    movel(p[x_c + 0.055265, y_c + -0.106909, z_c, rx, ry, rz], a, v)
    movel(p[x_c + 0.055232, y_c + -0.106894, z_c, rx, ry, rz], a, v)
    movel(p[x_c + 0.055195, y_c + -0.106876, z_c, rx, ry, rz], a, v)
    movel(p[x_c + 0.055155, y_c + -0.106856, z_c, rx, ry, rz], a, v)
    movel(p[x_c + 0.055111, y_c + -0.106832, z_c, rx, ry, rz], a, v)
    movel(p[x_c + 0.055063, y_c + -0.106806, z_c, rx, ry, rz], a, v)
    movel(p[x_c + 0.055012, y_c + -0.106778, z_c, rx, ry, rz], a, v)
    movel(p[x_c + 0.054956, y_c + -0.106746, z_c, rx, ry, rz], a, v)
    movel(p[x_c + 0.054897, y_c + -0.106712, z_c, rx, ry, rz], a, v)
    movel(p[x_c + 0.054834, y_c + -0.106675, z_c, rx, ry, rz], a, v)
    movel(p[x_c + 0.054767, y_c + -0.106635, z_c, rx, ry, rz], a, v)
    movel(p[x_c + 0.054696, y_c + -0.106592, z_c, rx, ry, rz], a, v)
    movel(p[x_c + 0.054696, y_c + -0.106592, z_c, rx, ry, rz], a, v)
    movel(p[x_c + 0.054632, y_c + -0.106555, z_c, rx, ry, rz], a, v)
    movel(p[x_c + 0.054557, y_c + -0.106511, z_c, rx, ry, rz], a, v)
    movel(p[x_c + 0.054470, y_c + -0.106462, z_c, rx, ry, rz], a, v)
    movel(p[x_c + 0.054372, y_c + -0.106408, z_c, rx, ry, rz], a, v)
    movel(p[x_c + 0.054263, y_c + -0.106348, z_c, rx, ry, rz], a, v)
    movel(p[x_c + 0.054144, y_c + -0.106284, z_c, rx, ry, rz], a, v)
    movel(p[x_c + 0.054016, y_c + -0.106215, z_c, rx, ry, rz], a, v)
    movel(p[x_c + 0.053879, y_c + -0.106142, z_c, rx, ry, rz], a, v)
    movel(p[x_c + 0.053733, y_c + -0.106065, z_c, rx, ry, rz], a, v)
    movel(p[x_c + 0.053580, y_c + -0.105984, z_c, rx, ry, rz], a, v)
    movel(p[x_c + 0.053420, y_c + -0.105900, z_c, rx, ry, rz], a, v)
    movel(p[x_c + 0.053253, y_c + -0.105813, z_c, rx, ry, rz], a, v)
    movel(p[x_c + 0.053080, y_c + -0.105722, z_c, rx, ry, rz], a, v)
    movel(p[x_c + 0.052901, y_c + -0.105630, z_c, rx, ry, rz], a, v)
    movel(p[x_c + 0.052717, y_c + -0.105535, z_c, rx, ry, rz], a, v)
    movel(p[x_c + 0.052529, y_c + -0.105438, z_c, rx, ry, rz], a, v)
    movel(p[x_c + 0.052338, y_c + -0.105339, z_c, rx, ry, rz], a, v)
    movel(p[x_c + 0.052143, y_c + -0.105239, z_c, rx, ry, rz], a, v)
    movel(p[x_c + 0.051945, y_c + -0.105138, z_c, rx, ry, rz], a, v)
    movel(p[x_c + 0.051745, y_c + -0.105036, z_c, rx, ry, rz], a, v)
    movel(p[x_c + 0.051543, y_c + -0.104933, z_c, rx, ry, rz], a, v)
    movel(p[x_c + 0.051341, y_c + -0.104830, z_c, rx, ry, rz], a, v)
    movel(p[x_c + 0.051138, y_c + -0.104727, z_c, rx, ry, rz], a, v)
    movel(p[x_c + 0.050935, y_c + -0.104625, z_c, rx, ry, rz], a, v)
    movel(p[x_c + 0.050733, y_c + -0.104523, z_c, rx, ry, rz], a, v)
    movel(p[x_c + 0.050532, y_c + -0.104421, z_c, rx, ry, rz], a, v)
    movel(p[x_c + 0.050332, y_c + -0.104321, z_c, rx, ry, rz], a, v)
    movel(p[x_c + 0.050135, y_c + -0.104222, z_c, rx, ry, rz], a, v)
    movel(p[x_c + 0.049941, y_c + -0.104125, z_c, rx, ry, rz], a, v)
    movel(p[x_c + 0.049751, y_c + -0.104030, z_c, rx, ry, rz], a, v)
    movel(p[x_c + 0.049564, y_c + -0.103938, z_c, rx, ry, rz], a, v)
    movel(p[x_c + 0.049382, y_c + -0.103847, z_c, rx, ry, rz], a, v)
    movel(p[x_c + 0.049205, y_c + -0.103760, z_c, rx, ry, rz], a, v)
    movel(p[x_c + 0.049034, y_c + -0.103676, z_c, rx, ry, rz], a, v)
    movel(p[x_c + 0.048869, y_c + -0.103595, z_c, rx, ry, rz], a, v)
    movel(p[x_c + 0.048711, y_c + -0.103517, z_c, rx, ry, rz], a, v)
    movel(p[x_c + 0.048560, y_c + -0.103444, z_c, rx, ry, rz], a, v)
    movel(p[x_c + 0.048417, y_c + -0.103375, z_c, rx, ry, rz], a, v)
    movel(p[x_c + 0.048283, y_c + -0.103310, z_c, rx, ry, rz], a, v)
    movel(p[x_c + 0.048158, y_c + -0.103251, z_c, rx, ry, rz], a, v)
    movel(p[x_c + 0.048042, y_c + -0.103196, z_c, rx, ry, rz], a, v)
    movel(p[x_c + 0.047937, y_c + -0.103147, z_c, rx, ry, rz], a, v)
    movel(p[x_c + 0.047842, y_c + -0.103103, z_c, rx, ry, rz], a, v)
    movel(p[x_c + 0.047759, y_c + -0.103065, z_c, rx, ry, rz], a, v)
    movel(p[x_c + 0.047687, y_c + -0.103034, z_c, rx, ry, rz], a, v)
    movel(p[x_c + 0.047628, y_c + -0.103009, z_c, rx, ry, rz], a, v)
    movel(p[x_c + 0.047582, y_c + -0.102991, z_c, rx, ry, rz], a, v)
    movel(p[x_c + 0.047550, y_c + -0.102980, z_c, rx, ry, rz], a, v)
    movel(p[x_c + 0.047531, y_c + -0.102976, z_c, rx, ry, rz], a, v)
    movel(p[x_c + 0.047531, y_c + -0.102976, z_c, rx, ry, rz], a, v)
    movel(p[x_c + 0.047525, y_c + -0.102977, z_c, rx, ry, rz], a, v)
    movel(p[x_c + 0.047514, y_c + -0.102981, z_c, rx, ry, rz], a, v)
    movel(p[x_c + 0.047501, y_c + -0.102987, z_c, rx, ry, rz], a, v)
    movel(p[x_c + 0.047483, y_c + -0.102996, z_c, rx, ry, rz], a, v)
    movel(p[x_c + 0.047462, y_c + -0.103007, z_c, rx, ry, rz], a, v)
    movel(p[x_c + 0.047437, y_c + -0.103020, z_c, rx, ry, rz], a, v)
    movel(p[x_c + 0.047409, y_c + -0.103036, z_c, rx, ry, rz], a, v)
    movel(p[x_c + 0.047378, y_c + -0.103054, z_c, rx, ry, rz], a, v)
    movel(p[x_c + 0.047343, y_c + -0.103074, z_c, rx, ry, rz], a, v)
    movel(p[x_c + 0.047306, y_c + -0.103097, z_c, rx, ry, rz], a, v)
    movel(p[x_c + 0.047265, y_c + -0.103121, z_c, rx, ry, rz], a, v)
    movel(p[x_c + 0.047220, y_c + -0.103148, z_c, rx, ry, rz], a, v)
    movel(p[x_c + 0.047173, y_c + -0.103177, z_c, rx, ry, rz], a, v)
    movel(p[x_c + 0.047123, y_c + -0.103207, z_c, rx, ry, rz], a, v)
    movel(p[x_c + 0.047070, y_c + -0.103240, z_c, rx, ry, rz], a, v)
    movel(p[x_c + 0.047014, y_c + -0.103275, z_c, rx, ry, rz], a, v)
    movel(p[x_c + 0.046956, y_c + -0.103311, z_c, rx, ry, rz], a, v)
    movel(p[x_c + 0.046894, y_c + -0.103350, z_c, rx, ry, rz], a, v)
    movel(p[x_c + 0.046830, y_c + -0.103390, z_c, rx, ry, rz], a, v)
    movel(p[x_c + 0.046763, y_c + -0.103432, z_c, rx, ry, rz], a, v)
    movel(p[x_c + 0.046694, y_c + -0.103476, z_c, rx, ry, rz], a, v)
    movel(p[x_c + 0.046623, y_c + -0.103521, z_c, rx, ry, rz], a, v)
    movel(p[x_c + 0.046548, y_c + -0.103568, z_c, rx, ry, rz], a, v)
    movel(p[x_c + 0.046472, y_c + -0.103617, z_c, rx, ry, rz], a, v)
    movel(p[x_c + 0.046393, y_c + -0.103667, z_c, rx, ry, rz], a, v)
    movel(p[x_c + 0.046312, y_c + -0.103719, z_c, rx, ry, rz], a, v)
    movel(p[x_c + 0.046229, y_c + -0.103773, z_c, rx, ry, rz], a, v)
    movel(p[x_c + 0.046144, y_c + -0.103827, z_c, rx, ry, rz], a, v)
    movel(p[x_c + 0.046057, y_c + -0.103884, z_c, rx, ry, rz], a, v)
    movel(p[x_c + 0.045968, y_c + -0.103941, z_c, rx, ry, rz], a, v)
    movel(p[x_c + 0.045877, y_c + -0.104000, z_c, rx, ry, rz], a, v)
    movel(p[x_c + 0.045784, y_c + -0.104061, z_c, rx, ry, rz], a, v)
    movel(p[x_c + 0.045689, y_c + -0.104122, z_c, rx, ry, rz], a, v)
    movel(p[x_c + 0.045593, y_c + -0.104185, z_c, rx, ry, rz], a, v)
    movel(p[x_c + 0.045495, y_c + -0.104249, z_c, rx, ry, rz], a, v)
    movel(p[x_c + 0.045395, y_c + -0.104314, z_c, rx, ry, rz], a, v)
    movel(p[x_c + 0.045294, y_c + -0.104380, z_c, rx, ry, rz], a, v)
    movel(p[x_c + 0.045191, y_c + -0.104447, z_c, rx, ry, rz], a, v)
    movel(p[x_c + 0.045088, y_c + -0.104515, z_c, rx, ry, rz], a, v)
    movel(p[x_c + 0.044982, y_c + -0.104584, z_c, rx, ry, rz], a, v)
    movel(p[x_c + 0.044876, y_c + -0.104654, z_c, rx, ry, rz], a, v)
    movel(p[x_c + 0.044768, y_c + -0.104725, z_c, rx, ry, rz], a, v)
    movel(p[x_c + 0.044659, y_c + -0.104797, z_c, rx, ry, rz], a, v)
    movel(p[x_c + 0.044549, y_c + -0.104870, z_c, rx, ry, rz], a, v)
    movel(p[x_c + 0.044438, y_c + -0.104943, z_c, rx, ry, rz], a, v)
    movel(p[x_c + 0.044326, y_c + -0.105017, z_c, rx, ry, rz], a, v)
    movel(p[x_c + 0.044213, y_c + -0.105092, z_c, rx, ry, rz], a, v)
    movel(p[x_c + 0.044099, y_c + -0.105168, z_c, rx, ry, rz], a, v)
    movel(p[x_c + 0.043985, y_c + -0.105244, z_c, rx, ry, rz], a, v)
    movel(p[x_c + 0.043985, y_c + -0.105244, z_c, rx, ry, rz], a, v)
    movel(p[x_c + 0.043855, y_c + -0.105330, z_c, rx, ry, rz], a, v)
    movel(p[x_c + 0.043724, y_c + -0.105416, z_c, rx, ry, rz], a, v)
    movel(p[x_c + 0.043591, y_c + -0.105503, z_c, rx, ry, rz], a, v)
    movel(p[x_c + 0.043457, y_c + -0.105590, z_c, rx, ry, rz], a, v)
    movel(p[x_c + 0.043321, y_c + -0.105677, z_c, rx, ry, rz], a, v)
    movel(p[x_c + 0.043184, y_c + -0.105765, z_c, rx, ry, rz], a, v)
    movel(p[x_c + 0.043045, y_c + -0.105853, z_c, rx, ry, rz], a, v)
    movel(p[x_c + 0.042905, y_c + -0.105941, z_c, rx, ry, rz], a, v)
    movel(p[x_c + 0.042764, y_c + -0.106030, z_c, rx, ry, rz], a, v)
    movel(p[x_c + 0.042622, y_c + -0.106119, z_c, rx, ry, rz], a, v)
    movel(p[x_c + 0.042478, y_c + -0.106207, z_c, rx, ry, rz], a, v)
    movel(p[x_c + 0.042334, y_c + -0.106296, z_c, rx, ry, rz], a, v)
    movel(p[x_c + 0.042188, y_c + -0.106385, z_c, rx, ry, rz], a, v)
    movel(p[x_c + 0.042042, y_c + -0.106474, z_c, rx, ry, rz], a, v)
    movel(p[x_c + 0.041894, y_c + -0.106563, z_c, rx, ry, rz], a, v)
    movel(p[x_c + 0.041746, y_c + -0.106652, z_c, rx, ry, rz], a, v)
    movel(p[x_c + 0.041597, y_c + -0.106741, z_c, rx, ry, rz], a, v)
    movel(p[x_c + 0.041447, y_c + -0.106830, z_c, rx, ry, rz], a, v)
    movel(p[x_c + 0.041296, y_c + -0.106919, z_c, rx, ry, rz], a, v)
    movel(p[x_c + 0.041145, y_c + -0.107007, z_c, rx, ry, rz], a, v)
    movel(p[x_c + 0.040994, y_c + -0.107096, z_c, rx, ry, rz], a, v)
    movel(p[x_c + 0.040841, y_c + -0.107184, z_c, rx, ry, rz], a, v)
    movel(p[x_c + 0.040688, y_c + -0.107272, z_c, rx, ry, rz], a, v)
    movel(p[x_c + 0.040535, y_c + -0.107360, z_c, rx, ry, rz], a, v)
    movel(p[x_c + 0.040382, y_c + -0.107447, z_c, rx, ry, rz], a, v)
    movel(p[x_c + 0.040228, y_c + -0.107535, z_c, rx, ry, rz], a, v)
    movel(p[x_c + 0.040074, y_c + -0.107621, z_c, rx, ry, rz], a, v)
    movel(p[x_c + 0.039919, y_c + -0.107708, z_c, rx, ry, rz], a, v)
    movel(p[x_c + 0.039765, y_c + -0.107794, z_c, rx, ry, rz], a, v)
    movel(p[x_c + 0.039610, y_c + -0.107879, z_c, rx, ry, rz], a, v)
    movel(p[x_c + 0.039456, y_c + -0.107964, z_c, rx, ry, rz], a, v)
    movel(p[x_c + 0.039301, y_c + -0.108049, z_c, rx, ry, rz], a, v)
    movel(p[x_c + 0.039147, y_c + -0.108133, z_c, rx, ry, rz], a, v)
    movel(p[x_c + 0.038992, y_c + -0.108216, z_c, rx, ry, rz], a, v)
    movel(p[x_c + 0.038838, y_c + -0.108299, z_c, rx, ry, rz], a, v)
    movel(p[x_c + 0.038684, y_c + -0.108381, z_c, rx, ry, rz], a, v)
    movel(p[x_c + 0.038531, y_c + -0.108463, z_c, rx, ry, rz], a, v)
    movel(p[x_c + 0.038377, y_c + -0.108543, z_c, rx, ry, rz], a, v)
    movel(p[x_c + 0.038224, y_c + -0.108623, z_c, rx, ry, rz], a, v)
    movel(p[x_c + 0.038072, y_c + -0.108703, z_c, rx, ry, rz], a, v)
    movel(p[x_c + 0.037920, y_c + -0.108781, z_c, rx, ry, rz], a, v)
    movel(p[x_c + 0.037769, y_c + -0.108859, z_c, rx, ry, rz], a, v)
    movel(p[x_c + 0.037618, y_c + -0.108936, z_c, rx, ry, rz], a, v)
    movel(p[x_c + 0.037468, y_c + -0.109012, z_c, rx, ry, rz], a, v)
    movel(p[x_c + 0.037318, y_c + -0.109087, z_c, rx, ry, rz], a, v)
    movel(p[x_c + 0.037170, y_c + -0.109161, z_c, rx, ry, rz], a, v)
    movel(p[x_c + 0.037022, y_c + -0.109234, z_c, rx, ry, rz], a, v)
    movel(p[x_c + 0.036875, y_c + -0.109306, z_c, rx, ry, rz], a, v)
    movel(p[x_c + 0.036729, y_c + -0.109377, z_c, rx, ry, rz], a, v)
    movel(p[x_c + 0.036729, y_c + -0.109377, z_c, rx, ry, rz], a, v)
    movel(p[x_c + 0.036600, y_c + -0.109440, z_c, rx, ry, rz], a, v)
    movel(p[x_c + 0.036471, y_c + -0.109503, z_c, rx, ry, rz], a, v)
    movel(p[x_c + 0.036342, y_c + -0.109567, z_c, rx, ry, rz], a, v)
    movel(p[x_c + 0.036213, y_c + -0.109630, z_c, rx, ry, rz], a, v)
    movel(p[x_c + 0.036085, y_c + -0.109694, z_c, rx, ry, rz], a, v)
    movel(p[x_c + 0.035957, y_c + -0.109757, z_c, rx, ry, rz], a, v)
    movel(p[x_c + 0.035830, y_c + -0.109821, z_c, rx, ry, rz], a, v)
    movel(p[x_c + 0.035704, y_c + -0.109885, z_c, rx, ry, rz], a, v)
    movel(p[x_c + 0.035578, y_c + -0.109948, z_c, rx, ry, rz], a, v)
    movel(p[x_c + 0.035453, y_c + -0.110012, z_c, rx, ry, rz], a, v)
    movel(p[x_c + 0.035329, y_c + -0.110075, z_c, rx, ry, rz], a, v)
    movel(p[x_c + 0.035206, y_c + -0.110138, z_c, rx, ry, rz], a, v)
    movel(p[x_c + 0.035085, y_c + -0.110201, z_c, rx, ry, rz], a, v)
    movel(p[x_c + 0.034964, y_c + -0.110263, z_c, rx, ry, rz], a, v)
    movel(p[x_c + 0.034845, y_c + -0.110325, z_c, rx, ry, rz], a, v)
    movel(p[x_c + 0.034727, y_c + -0.110387, z_c, rx, ry, rz], a, v)
    movel(p[x_c + 0.034610, y_c + -0.110448, z_c, rx, ry, rz], a, v)
    movel(p[x_c + 0.034495, y_c + -0.110509, z_c, rx, ry, rz], a, v)
    movel(p[x_c + 0.034382, y_c + -0.110570, z_c, rx, ry, rz], a, v)
    movel(p[x_c + 0.034270, y_c + -0.110629, z_c, rx, ry, rz], a, v)
    movel(p[x_c + 0.034160, y_c + -0.110688, z_c, rx, ry, rz], a, v)
    movel(p[x_c + 0.034052, y_c + -0.110747, z_c, rx, ry, rz], a, v)
    movel(p[x_c + 0.033946, y_c + -0.110804, z_c, rx, ry, rz], a, v)
    movel(p[x_c + 0.033841, y_c + -0.110861, z_c, rx, ry, rz], a, v)
    movel(p[x_c + 0.033739, y_c + -0.110918, z_c, rx, ry, rz], a, v)
    movel(p[x_c + 0.033639, y_c + -0.110973, z_c, rx, ry, rz], a, v)
    movel(p[x_c + 0.033541, y_c + -0.111027, z_c, rx, ry, rz], a, v)
    movel(p[x_c + 0.033446, y_c + -0.111081, z_c, rx, ry, rz], a, v)
    movel(p[x_c + 0.033353, y_c + -0.111133, z_c, rx, ry, rz], a, v)
    movel(p[x_c + 0.033262, y_c + -0.111185, z_c, rx, ry, rz], a, v)
    movel(p[x_c + 0.033174, y_c + -0.111235, z_c, rx, ry, rz], a, v)
    movel(p[x_c + 0.033089, y_c + -0.111284, z_c, rx, ry, rz], a, v)
    movel(p[x_c + 0.033007, y_c + -0.111332, z_c, rx, ry, rz], a, v)
    movel(p[x_c + 0.032927, y_c + -0.111379, z_c, rx, ry, rz], a, v)
    movel(p[x_c + 0.032850, y_c + -0.111425, z_c, rx, ry, rz], a, v)
    movel(p[x_c + 0.032776, y_c + -0.111469, z_c, rx, ry, rz], a, v)
    movel(p[x_c + 0.032705, y_c + -0.111512, z_c, rx, ry, rz], a, v)
    movel(p[x_c + 0.032638, y_c + -0.111554, z_c, rx, ry, rz], a, v)
    movel(p[x_c + 0.032573, y_c + -0.111594, z_c, rx, ry, rz], a, v)
    movel(p[x_c + 0.032512, y_c + -0.111633, z_c, rx, ry, rz], a, v)
    movel(p[x_c + 0.032455, y_c + -0.111670, z_c, rx, ry, rz], a, v)
    movel(p[x_c + 0.032400, y_c + -0.111706, z_c, rx, ry, rz], a, v)
    movel(p[x_c + 0.032350, y_c + -0.111739, z_c, rx, ry, rz], a, v)
    movel(p[x_c + 0.032303, y_c + -0.111772, z_c, rx, ry, rz], a, v)
    movel(p[x_c + 0.032259, y_c + -0.111802, z_c, rx, ry, rz], a, v)
    movel(p[x_c + 0.032220, y_c + -0.111831, z_c, rx, ry, rz], a, v)
    movel(p[x_c + 0.032184, y_c + -0.111858, z_c, rx, ry, rz], a, v)
    movel(p[x_c + 0.032153, y_c + -0.111884, z_c, rx, ry, rz], a, v)
    movel(p[x_c + 0.032125, y_c + -0.111907, z_c, rx, ry, rz], a, v)
    movel(p[x_c + 0.032125, y_c + -0.111907, z_c, rx, ry, rz], a, v)
    movel(p[x_c + 0.032099, y_c + -0.111931, z_c, rx, ry, rz], a, v)
    movel(p[x_c + 0.032070, y_c + -0.111957, z_c, rx, ry, rz], a, v)
    movel(p[x_c + 0.032040, y_c + -0.111986, z_c, rx, ry, rz], a, v)
    movel(p[x_c + 0.032008, y_c + -0.112018, z_c, rx, ry, rz], a, v)
    movel(p[x_c + 0.031974, y_c + -0.112053, z_c, rx, ry, rz], a, v)
    movel(p[x_c + 0.031939, y_c + -0.112089, z_c, rx, ry, rz], a, v)
    movel(p[x_c + 0.031902, y_c + -0.112129, z_c, rx, ry, rz], a, v)
    movel(p[x_c + 0.031863, y_c + -0.112170, z_c, rx, ry, rz], a, v)
    movel(p[x_c + 0.031823, y_c + -0.112214, z_c, rx, ry, rz], a, v)
    movel(p[x_c + 0.031781, y_c + -0.112261, z_c, rx, ry, rz], a, v)
    movel(p[x_c + 0.031737, y_c + -0.112309, z_c, rx, ry, rz], a, v)
    movel(p[x_c + 0.031693, y_c + -0.112360, z_c, rx, ry, rz], a, v)
    movel(p[x_c + 0.031646, y_c + -0.112413, z_c, rx, ry, rz], a, v)
    movel(p[x_c + 0.031599, y_c + -0.112468, z_c, rx, ry, rz], a, v)
    movel(p[x_c + 0.031550, y_c + -0.112524, z_c, rx, ry, rz], a, v)
    movel(p[x_c + 0.031500, y_c + -0.112583, z_c, rx, ry, rz], a, v)
    movel(p[x_c + 0.031449, y_c + -0.112644, z_c, rx, ry, rz], a, v)
    movel(p[x_c + 0.031396, y_c + -0.112706, z_c, rx, ry, rz], a, v)
    movel(p[x_c + 0.031343, y_c + -0.112770, z_c, rx, ry, rz], a, v)
    movel(p[x_c + 0.031289, y_c + -0.112836, z_c, rx, ry, rz], a, v)
    movel(p[x_c + 0.031233, y_c + -0.112903, z_c, rx, ry, rz], a, v)
    movel(p[x_c + 0.031177, y_c + -0.112972, z_c, rx, ry, rz], a, v)
    movel(p[x_c + 0.031119, y_c + -0.113043, z_c, rx, ry, rz], a, v)
    movel(p[x_c + 0.031061, y_c + -0.113114, z_c, rx, ry, rz], a, v)
    movel(p[x_c + 0.031002, y_c + -0.113188, z_c, rx, ry, rz], a, v)
    movel(p[x_c + 0.030942, y_c + -0.113262, z_c, rx, ry, rz], a, v)
    movel(p[x_c + 0.030882, y_c + -0.113338, z_c, rx, ry, rz], a, v)
    movel(p[x_c + 0.030820, y_c + -0.113415, z_c, rx, ry, rz], a, v)
    movel(p[x_c + 0.030759, y_c + -0.113494, z_c, rx, ry, rz], a, v)
    movel(p[x_c + 0.030696, y_c + -0.113573, z_c, rx, ry, rz], a, v)
    movel(p[x_c + 0.030633, y_c + -0.113653, z_c, rx, ry, rz], a, v)
    movel(p[x_c + 0.030570, y_c + -0.113735, z_c, rx, ry, rz], a, v)
    movel(p[x_c + 0.030506, y_c + -0.113817, z_c, rx, ry, rz], a, v)
    movel(p[x_c + 0.030442, y_c + -0.113900, z_c, rx, ry, rz], a, v)
    movel(p[x_c + 0.030377, y_c + -0.113984, z_c, rx, ry, rz], a, v)
    movel(p[x_c + 0.030312, y_c + -0.114069, z_c, rx, ry, rz], a, v)
    movel(p[x_c + 0.030247, y_c + -0.114154, z_c, rx, ry, rz], a, v)
    movel(p[x_c + 0.030182, y_c + -0.114240, z_c, rx, ry, rz], a, v)
    movel(p[x_c + 0.030117, y_c + -0.114326, z_c, rx, ry, rz], a, v)
    movel(p[x_c + 0.030051, y_c + -0.114413, z_c, rx, ry, rz], a, v)
    movel(p[x_c + 0.029986, y_c + -0.114501, z_c, rx, ry, rz], a, v)
    movel(p[x_c + 0.029920, y_c + -0.114588, z_c, rx, ry, rz], a, v)
    movel(p[x_c + 0.029855, y_c + -0.114677, z_c, rx, ry, rz], a, v)
    movel(p[x_c + 0.029789, y_c + -0.114765, z_c, rx, ry, rz], a, v)
    movel(p[x_c + 0.029724, y_c + -0.114854, z_c, rx, ry, rz], a, v)
    movel(p[x_c + 0.029659, y_c + -0.114942, z_c, rx, ry, rz], a, v)
    movel(p[x_c + 0.029594, y_c + -0.115031, z_c, rx, ry, rz], a, v)
    movel(p[x_c + 0.029529, y_c + -0.115120, z_c, rx, ry, rz], a, v)
    movel(p[x_c + 0.029465, y_c + -0.115209, z_c, rx, ry, rz], a, v)
    movel(p[x_c + 0.029465, y_c + -0.115209, z_c, rx, ry, rz], a, v)
    movel(p[x_c + 0.029321, y_c + -0.115407, z_c, rx, ry, rz], a, v)
    movel(p[x_c + 0.029177, y_c + -0.115603, z_c, rx, ry, rz], a, v)
    movel(p[x_c + 0.029032, y_c + -0.115797, z_c, rx, ry, rz], a, v)
    movel(p[x_c + 0.028888, y_c + -0.115988, z_c, rx, ry, rz], a, v)
    movel(p[x_c + 0.028743, y_c + -0.116177, z_c, rx, ry, rz], a, v)
    movel(p[x_c + 0.028599, y_c + -0.116363, z_c, rx, ry, rz], a, v)
    movel(p[x_c + 0.028454, y_c + -0.116547, z_c, rx, ry, rz], a, v)
    movel(p[x_c + 0.028309, y_c + -0.116728, z_c, rx, ry, rz], a, v)
    movel(p[x_c + 0.028165, y_c + -0.116907, z_c, rx, ry, rz], a, v)
    movel(p[x_c + 0.028020, y_c + -0.117083, z_c, rx, ry, rz], a, v)
    movel(p[x_c + 0.027875, y_c + -0.117257, z_c, rx, ry, rz], a, v)
    movel(p[x_c + 0.027730, y_c + -0.117428, z_c, rx, ry, rz], a, v)
    movel(p[x_c + 0.027586, y_c + -0.117597, z_c, rx, ry, rz], a, v)
    movel(p[x_c + 0.027441, y_c + -0.117763, z_c, rx, ry, rz], a, v)
    movel(p[x_c + 0.027296, y_c + -0.117926, z_c, rx, ry, rz], a, v)
    movel(p[x_c + 0.027152, y_c + -0.118087, z_c, rx, ry, rz], a, v)
    movel(p[x_c + 0.027007, y_c + -0.118245, z_c, rx, ry, rz], a, v)
    movel(p[x_c + 0.026863, y_c + -0.118401, z_c, rx, ry, rz], a, v)
    movel(p[x_c + 0.026719, y_c + -0.118554, z_c, rx, ry, rz], a, v)
    movel(p[x_c + 0.026574, y_c + -0.118704, z_c, rx, ry, rz], a, v)
    movel(p[x_c + 0.026430, y_c + -0.118852, z_c, rx, ry, rz], a, v)
    movel(p[x_c + 0.026287, y_c + -0.118997, z_c, rx, ry, rz], a, v)
    movel(p[x_c + 0.026143, y_c + -0.119139, z_c, rx, ry, rz], a, v)
    movel(p[x_c + 0.025999, y_c + -0.119279, z_c, rx, ry, rz], a, v)
    movel(p[x_c + 0.025856, y_c + -0.119415, z_c, rx, ry, rz], a, v)
    movel(p[x_c + 0.025713, y_c + -0.119550, z_c, rx, ry, rz], a, v)
    movel(p[x_c + 0.025570, y_c + -0.119681, z_c, rx, ry, rz], a, v)
    movel(p[x_c + 0.025427, y_c + -0.119810, z_c, rx, ry, rz], a, v)
    movel(p[x_c + 0.025284, y_c + -0.119936, z_c, rx, ry, rz], a, v)
    movel(p[x_c + 0.025142, y_c + -0.120059, z_c, rx, ry, rz], a, v)
    movel(p[x_c + 0.025000, y_c + -0.120179, z_c, rx, ry, rz], a, v)
    movel(p[x_c + 0.024859, y_c + -0.120297, z_c, rx, ry, rz], a, v)
    movel(p[x_c + 0.024717, y_c + -0.120412, z_c, rx, ry, rz], a, v)
    movel(p[x_c + 0.024576, y_c + -0.120524, z_c, rx, ry, rz], a, v)
    movel(p[x_c + 0.024435, y_c + -0.120633, z_c, rx, ry, rz], a, v)
    movel(p[x_c + 0.024295, y_c + -0.120739, z_c, rx, ry, rz], a, v)
    movel(p[x_c + 0.024155, y_c + -0.120842, z_c, rx, ry, rz], a, v)
    movel(p[x_c + 0.024015, y_c + -0.120943, z_c, rx, ry, rz], a, v)
    movel(p[x_c + 0.023875, y_c + -0.121041, z_c, rx, ry, rz], a, v)
    movel(p[x_c + 0.023736, y_c + -0.121135, z_c, rx, ry, rz], a, v)
    movel(p[x_c + 0.023598, y_c + -0.121227, z_c, rx, ry, rz], a, v)
    movel(p[x_c + 0.023459, y_c + -0.121316, z_c, rx, ry, rz], a, v)
    movel(p[x_c + 0.023322, y_c + -0.121402, z_c, rx, ry, rz], a, v)
    movel(p[x_c + 0.023184, y_c + -0.121485, z_c, rx, ry, rz], a, v)
    movel(p[x_c + 0.023047, y_c + -0.121565, z_c, rx, ry, rz], a, v)
    movel(p[x_c + 0.022911, y_c + -0.121642, z_c, rx, ry, rz], a, v)
    movel(p[x_c + 0.022775, y_c + -0.121716, z_c, rx, ry, rz], a, v)
    movel(p[x_c + 0.022639, y_c + -0.121788, z_c, rx, ry, rz], a, v)
    movel(p[x_c + 0.022504, y_c + -0.121856, z_c, rx, ry, rz], a, v)
    movel(p[x_c + 0.022504, y_c + -0.121856, z_c, rx, ry, rz], a, v)
    movel(p[x_c + 0.020881, y_c + -0.122658, z_c, rx, ry, rz], a, v)
    movel(p[x_c + 0.020881, y_c + -0.122658, z_c, rx, ry, rz], a, v)
    movel(p[x_c + 0.018590, y_c + -0.122275, z_c, rx, ry, rz], a, v)
    movel(p[x_c + 0.018590, y_c + -0.122275, z_c, rx, ry, rz], a, v)
    movel(p[x_c + 0.018405, y_c + -0.122244, z_c, rx, ry, rz], a, v)
    movel(p[x_c + 0.018222, y_c + -0.122216, z_c, rx, ry, rz], a, v)
    movel(p[x_c + 0.018040, y_c + -0.122189, z_c, rx, ry, rz], a, v)
    movel(p[x_c + 0.017859, y_c + -0.122164, z_c, rx, ry, rz], a, v)
    movel(p[x_c + 0.017680, y_c + -0.122140, z_c, rx, ry, rz], a, v)
    movel(p[x_c + 0.017502, y_c + -0.122118, z_c, rx, ry, rz], a, v)
    movel(p[x_c + 0.017326, y_c + -0.122098, z_c, rx, ry, rz], a, v)
    movel(p[x_c + 0.017150, y_c + -0.122080, z_c, rx, ry, rz], a, v)
    movel(p[x_c + 0.016976, y_c + -0.122063, z_c, rx, ry, rz], a, v)
    movel(p[x_c + 0.016802, y_c + -0.122048, z_c, rx, ry, rz], a, v)
    movel(p[x_c + 0.016630, y_c + -0.122034, z_c, rx, ry, rz], a, v)
    movel(p[x_c + 0.016458, y_c + -0.122023, z_c, rx, ry, rz], a, v)
    movel(p[x_c + 0.016287, y_c + -0.122013, z_c, rx, ry, rz], a, v)
    movel(p[x_c + 0.016117, y_c + -0.122005, z_c, rx, ry, rz], a, v)
    movel(p[x_c + 0.015947, y_c + -0.121998, z_c, rx, ry, rz], a, v)
    movel(p[x_c + 0.015778, y_c + -0.121993, z_c, rx, ry, rz], a, v)
    movel(p[x_c + 0.015610, y_c + -0.121990, z_c, rx, ry, rz], a, v)
    movel(p[x_c + 0.015441, y_c + -0.121989, z_c, rx, ry, rz], a, v)
    movel(p[x_c + 0.015274, y_c + -0.121989, z_c, rx, ry, rz], a, v)
    movel(p[x_c + 0.015106, y_c + -0.121991, z_c, rx, ry, rz], a, v)
    movel(p[x_c + 0.014939, y_c + -0.121995, z_c, rx, ry, rz], a, v)
    movel(p[x_c + 0.014772, y_c + -0.122001, z_c, rx, ry, rz], a, v)
    movel(p[x_c + 0.014605, y_c + -0.122008, z_c, rx, ry, rz], a, v)
    movel(p[x_c + 0.014438, y_c + -0.122018, z_c, rx, ry, rz], a, v)
    movel(p[x_c + 0.014270, y_c + -0.122028, z_c, rx, ry, rz], a, v)
    movel(p[x_c + 0.014103, y_c + -0.122041, z_c, rx, ry, rz], a, v)
    movel(p[x_c + 0.013936, y_c + -0.122056, z_c, rx, ry, rz], a, v)
    movel(p[x_c + 0.013768, y_c + -0.122072, z_c, rx, ry, rz], a, v)
    movel(p[x_c + 0.013600, y_c + -0.122090, z_c, rx, ry, rz], a, v)
    movel(p[x_c + 0.013431, y_c + -0.122110, z_c, rx, ry, rz], a, v)
    movel(p[x_c + 0.013262, y_c + -0.122131, z_c, rx, ry, rz], a, v)
    movel(p[x_c + 0.013093, y_c + -0.122155, z_c, rx, ry, rz], a, v)
    movel(p[x_c + 0.012923, y_c + -0.122180, z_c, rx, ry, rz], a, v)
    movel(p[x_c + 0.012752, y_c + -0.122207, z_c, rx, ry, rz], a, v)
    movel(p[x_c + 0.012580, y_c + -0.122236, z_c, rx, ry, rz], a, v)
    movel(p[x_c + 0.012408, y_c + -0.122267, z_c, rx, ry, rz], a, v)
    movel(p[x_c + 0.012234, y_c + -0.122299, z_c, rx, ry, rz], a, v)
    movel(p[x_c + 0.012060, y_c + -0.122333, z_c, rx, ry, rz], a, v)
    movel(p[x_c + 0.011885, y_c + -0.122370, z_c, rx, ry, rz], a, v)
    movel(p[x_c + 0.011708, y_c + -0.122408, z_c, rx, ry, rz], a, v)
    movel(p[x_c + 0.011530, y_c + -0.122447, z_c, rx, ry, rz], a, v)
    movel(p[x_c + 0.011351, y_c + -0.122489, z_c, rx, ry, rz], a, v)
    movel(p[x_c + 0.011171, y_c + -0.122533, z_c, rx, ry, rz], a, v)
    movel(p[x_c + 0.010989, y_c + -0.122578, z_c, rx, ry, rz], a, v)
    movel(p[x_c + 0.010806, y_c + -0.122625, z_c, rx, ry, rz], a, v)
    movel(p[x_c + 0.010622, y_c + -0.122674, z_c, rx, ry, rz], a, v)
    movel(p[x_c + 0.010435, y_c + -0.122725, z_c, rx, ry, rz], a, v)
    movel(p[x_c + 0.010247, y_c + -0.122778, z_c, rx, ry, rz], a, v)
    movel(p[x_c + 0.010057, y_c + -0.122833, z_c, rx, ry, rz], a, v)
    movel(p[x_c + 0.010057, y_c + -0.122833, z_c, rx, ry, rz], a, v)
    movel(p[x_c + 0.009819, y_c + -0.122902, z_c, rx, ry, rz], a, v)
    movel(p[x_c + 0.009585, y_c + -0.122969, z_c, rx, ry, rz], a, v)
    movel(p[x_c + 0.009357, y_c + -0.123034, z_c, rx, ry, rz], a, v)
    movel(p[x_c + 0.009133, y_c + -0.123097, z_c, rx, ry, rz], a, v)
    movel(p[x_c + 0.008913, y_c + -0.123157, z_c, rx, ry, rz], a, v)
    movel(p[x_c + 0.008697, y_c + -0.123216, z_c, rx, ry, rz], a, v)
    movel(p[x_c + 0.008485, y_c + -0.123272, z_c, rx, ry, rz], a, v)
    movel(p[x_c + 0.008277, y_c + -0.123327, z_c, rx, ry, rz], a, v)
    movel(p[x_c + 0.008071, y_c + -0.123380, z_c, rx, ry, rz], a, v)
    movel(p[x_c + 0.007869, y_c + -0.123430, z_c, rx, ry, rz], a, v)
    movel(p[x_c + 0.007668, y_c + -0.123479, z_c, rx, ry, rz], a, v)
    movel(p[x_c + 0.007471, y_c + -0.123526, z_c, rx, ry, rz], a, v)
    movel(p[x_c + 0.007275, y_c + -0.123571, z_c, rx, ry, rz], a, v)
    movel(p[x_c + 0.007080, y_c + -0.123615, z_c, rx, ry, rz], a, v)
    movel(p[x_c + 0.006887, y_c + -0.123656, z_c, rx, ry, rz], a, v)
    movel(p[x_c + 0.006695, y_c + -0.123696, z_c, rx, ry, rz], a, v)
    movel(p[x_c + 0.006504, y_c + -0.123735, z_c, rx, ry, rz], a, v)
    movel(p[x_c + 0.006313, y_c + -0.123771, z_c, rx, ry, rz], a, v)
    movel(p[x_c + 0.006122, y_c + -0.123807, z_c, rx, ry, rz], a, v)
    movel(p[x_c + 0.005932, y_c + -0.123840, z_c, rx, ry, rz], a, v)
    movel(p[x_c + 0.005740, y_c + -0.123873, z_c, rx, ry, rz], a, v)
    movel(p[x_c + 0.005548, y_c + -0.123904, z_c, rx, ry, rz], a, v)
    movel(p[x_c + 0.005355, y_c + -0.123933, z_c, rx, ry, rz], a, v)
    movel(p[x_c + 0.005161, y_c + -0.123961, z_c, rx, ry, rz], a, v)
    movel(p[x_c + 0.004965, y_c + -0.123988, z_c, rx, ry, rz], a, v)
    movel(p[x_c + 0.004767, y_c + -0.124014, z_c, rx, ry, rz], a, v)
    movel(p[x_c + 0.004567, y_c + -0.124038, z_c, rx, ry, rz], a, v)
    movel(p[x_c + 0.004364, y_c + -0.124061, z_c, rx, ry, rz], a, v)
    movel(p[x_c + 0.004159, y_c + -0.124083, z_c, rx, ry, rz], a, v)
    movel(p[x_c + 0.003950, y_c + -0.124104, z_c, rx, ry, rz], a, v)
    movel(p[x_c + 0.003738, y_c + -0.124124, z_c, rx, ry, rz], a, v)
    movel(p[x_c + 0.003522, y_c + -0.124143, z_c, rx, ry, rz], a, v)
    movel(p[x_c + 0.003303, y_c + -0.124161, z_c, rx, ry, rz], a, v)
    movel(p[x_c + 0.003079, y_c + -0.124177, z_c, rx, ry, rz], a, v)
    movel(p[x_c + 0.002850, y_c + -0.124193, z_c, rx, ry, rz], a, v)
    movel(p[x_c + 0.002617, y_c + -0.124209, z_c, rx, ry, rz], a, v)
    movel(p[x_c + 0.002378, y_c + -0.124223, z_c, rx, ry, rz], a, v)
    movel(p[x_c + 0.002134, y_c + -0.124236, z_c, rx, ry, rz], a, v)
    movel(p[x_c + 0.001884, y_c + -0.124249, z_c, rx, ry, rz], a, v)
    movel(p[x_c + 0.001628, y_c + -0.124261, z_c, rx, ry, rz], a, v)
    movel(p[x_c + 0.001365, y_c + -0.124273, z_c, rx, ry, rz], a, v)
    movel(p[x_c + 0.001096, y_c + -0.124284, z_c, rx, ry, rz], a, v)
    movel(p[x_c + 0.000820, y_c + -0.124294, z_c, rx, ry, rz], a, v)
    movel(p[x_c + 0.000537, y_c + -0.124304, z_c, rx, ry, rz], a, v)
    movel(p[x_c + 0.000246, y_c + -0.124313, z_c, rx, ry, rz], a, v)
    movel(p[x_c + -0.000053, y_c + -0.124322, z_c, rx, ry, rz], a, v)
    movel(p[x_c + -0.000360, y_c + -0.124330, z_c, rx, ry, rz], a, v)
    movel(p[x_c + -0.000675, y_c + -0.124338, z_c, rx, ry, rz], a, v)
    movel(p[x_c + -0.000999, y_c + -0.124346, z_c, rx, ry, rz], a, v)
    movel(p[x_c + -0.000999, y_c + -0.124346, z_c, rx, ry, rz], a, v)
    movel(p[x_c + -0.001227, y_c + -0.124351, z_c, rx, ry, rz], a, v)
    movel(p[x_c + -0.001452, y_c + -0.124355, z_c, rx, ry, rz], a, v)
    movel(p[x_c + -0.001674, y_c + -0.124360, z_c, rx, ry, rz], a, v)
    movel(p[x_c + -0.001893, y_c + -0.124364, z_c, rx, ry, rz], a, v)
    movel(p[x_c + -0.002109, y_c + -0.124367, z_c, rx, ry, rz], a, v)
    movel(p[x_c + -0.002322, y_c + -0.124370, z_c, rx, ry, rz], a, v)
    movel(p[x_c + -0.002532, y_c + -0.124373, z_c, rx, ry, rz], a, v)
    movel(p[x_c + -0.002741, y_c + -0.124375, z_c, rx, ry, rz], a, v)
    movel(p[x_c + -0.002946, y_c + -0.124376, z_c, rx, ry, rz], a, v)
    movel(p[x_c + -0.003150, y_c + -0.124378, z_c, rx, ry, rz], a, v)
    movel(p[x_c + -0.003352, y_c + -0.124379, z_c, rx, ry, rz], a, v)
    movel(p[x_c + -0.003551, y_c + -0.124379, z_c, rx, ry, rz], a, v)
    movel(p[x_c + -0.003749, y_c + -0.124379, z_c, rx, ry, rz], a, v)
    movel(p[x_c + -0.003946, y_c + -0.124379, z_c, rx, ry, rz], a, v)
    movel(p[x_c + -0.004140, y_c + -0.124378, z_c, rx, ry, rz], a, v)
    movel(p[x_c + -0.004334, y_c + -0.124376, z_c, rx, ry, rz], a, v)
    movel(p[x_c + -0.004526, y_c + -0.124374, z_c, rx, ry, rz], a, v)
    movel(p[x_c + -0.004717, y_c + -0.124372, z_c, rx, ry, rz], a, v)
    movel(p[x_c + -0.004907, y_c + -0.124369, z_c, rx, ry, rz], a, v)
    movel(p[x_c + -0.005096, y_c + -0.124366, z_c, rx, ry, rz], a, v)
    movel(p[x_c + -0.005285, y_c + -0.124362, z_c, rx, ry, rz], a, v)
    movel(p[x_c + -0.005473, y_c + -0.124358, z_c, rx, ry, rz], a, v)
    movel(p[x_c + -0.005660, y_c + -0.124353, z_c, rx, ry, rz], a, v)
    movel(p[x_c + -0.005847, y_c + -0.124348, z_c, rx, ry, rz], a, v)
    movel(p[x_c + -0.006034, y_c + -0.124342, z_c, rx, ry, rz], a, v)
    movel(p[x_c + -0.006221, y_c + -0.124336, z_c, rx, ry, rz], a, v)
    movel(p[x_c + -0.006409, y_c + -0.124329, z_c, rx, ry, rz], a, v)
    movel(p[x_c + -0.006596, y_c + -0.124322, z_c, rx, ry, rz], a, v)
    movel(p[x_c + -0.006784, y_c + -0.124314, z_c, rx, ry, rz], a, v)
    movel(p[x_c + -0.006972, y_c + -0.124306, z_c, rx, ry, rz], a, v)
    movel(p[x_c + -0.007161, y_c + -0.124297, z_c, rx, ry, rz], a, v)
    movel(p[x_c + -0.007350, y_c + -0.124288, z_c, rx, ry, rz], a, v)
    movel(p[x_c + -0.007541, y_c + -0.124278, z_c, rx, ry, rz], a, v)
    movel(p[x_c + -0.007732, y_c + -0.124268, z_c, rx, ry, rz], a, v)
    movel(p[x_c + -0.007925, y_c + -0.124257, z_c, rx, ry, rz], a, v)
    movel(p[x_c + -0.008119, y_c + -0.124245, z_c, rx, ry, rz], a, v)
    movel(p[x_c + -0.008315, y_c + -0.124233, z_c, rx, ry, rz], a, v)
    movel(p[x_c + -0.008512, y_c + -0.124221, z_c, rx, ry, rz], a, v)
    movel(p[x_c + -0.008710, y_c + -0.124208, z_c, rx, ry, rz], a, v)
    movel(p[x_c + -0.008911, y_c + -0.124194, z_c, rx, ry, rz], a, v)
    movel(p[x_c + -0.009114, y_c + -0.124180, z_c, rx, ry, rz], a, v)
    movel(p[x_c + -0.009318, y_c + -0.124165, z_c, rx, ry, rz], a, v)
    movel(p[x_c + -0.009525, y_c + -0.124150, z_c, rx, ry, rz], a, v)
    movel(p[x_c + -0.009734, y_c + -0.124134, z_c, rx, ry, rz], a, v)
    movel(p[x_c + -0.009946, y_c + -0.124117, z_c, rx, ry, rz], a, v)
    movel(p[x_c + -0.010161, y_c + -0.124100, z_c, rx, ry, rz], a, v)
    movel(p[x_c + -0.010378, y_c + -0.124082, z_c, rx, ry, rz], a, v)
    movel(p[x_c + -0.010598, y_c + -0.124064, z_c, rx, ry, rz], a, v)
    movel(p[x_c + -0.010821, y_c + -0.124045, z_c, rx, ry, rz], a, v)
    movel(p[x_c + -0.010821, y_c + -0.124045, z_c, rx, ry, rz], a, v)
    movel(p[x_c + -0.011304, y_c + -0.124005, z_c, rx, ry, rz], a, v)
    movel(p[x_c + -0.011785, y_c + -0.123966, z_c, rx, ry, rz], a, v)
    movel(p[x_c + -0.012264, y_c + -0.123930, z_c, rx, ry, rz], a, v)
    movel(p[x_c + -0.012739, y_c + -0.123896, z_c, rx, ry, rz], a, v)
    movel(p[x_c + -0.013213, y_c + -0.123863, z_c, rx, ry, rz], a, v)
    movel(p[x_c + -0.013683, y_c + -0.123833, z_c, rx, ry, rz], a, v)
    movel(p[x_c + -0.014150, y_c + -0.123804, z_c, rx, ry, rz], a, v)
    movel(p[x_c + -0.014615, y_c + -0.123777, z_c, rx, ry, rz], a, v)
    movel(p[x_c + -0.015075, y_c + -0.123753, z_c, rx, ry, rz], a, v)
    movel(p[x_c + -0.015533, y_c + -0.123730, z_c, rx, ry, rz], a, v)
    movel(p[x_c + -0.015986, y_c + -0.123709, z_c, rx, ry, rz], a, v)
    movel(p[x_c + -0.016436, y_c + -0.123690, z_c, rx, ry, rz], a, v)
    movel(p[x_c + -0.016882, y_c + -0.123673, z_c, rx, ry, rz], a, v)
    movel(p[x_c + -0.017323, y_c + -0.123658, z_c, rx, ry, rz], a, v)
    movel(p[x_c + -0.017760, y_c + -0.123645, z_c, rx, ry, rz], a, v)
    movel(p[x_c + -0.018193, y_c + -0.123634, z_c, rx, ry, rz], a, v)
    movel(p[x_c + -0.018621, y_c + -0.123624, z_c, rx, ry, rz], a, v)
    movel(p[x_c + -0.019043, y_c + -0.123617, z_c, rx, ry, rz], a, v)
    movel(p[x_c + -0.019461, y_c + -0.123612, z_c, rx, ry, rz], a, v)
    movel(p[x_c + -0.019874, y_c + -0.123608, z_c, rx, ry, rz], a, v)
    movel(p[x_c + -0.020281, y_c + -0.123606, z_c, rx, ry, rz], a, v)
    movel(p[x_c + -0.020683, y_c + -0.123607, z_c, rx, ry, rz], a, v)
    movel(p[x_c + -0.021079, y_c + -0.123609, z_c, rx, ry, rz], a, v)
    movel(p[x_c + -0.021468, y_c + -0.123613, z_c, rx, ry, rz], a, v)
    movel(p[x_c + -0.021852, y_c + -0.123619, z_c, rx, ry, rz], a, v)
    movel(p[x_c + -0.022230, y_c + -0.123627, z_c, rx, ry, rz], a, v)
    movel(p[x_c + -0.022601, y_c + -0.123637, z_c, rx, ry, rz], a, v)
    movel(p[x_c + -0.022966, y_c + -0.123648, z_c, rx, ry, rz], a, v)
    movel(p[x_c + -0.023323, y_c + -0.123662, z_c, rx, ry, rz], a, v)
    movel(p[x_c + -0.023674, y_c + -0.123677, z_c, rx, ry, rz], a, v)
    movel(p[x_c + -0.024018, y_c + -0.123694, z_c, rx, ry, rz], a, v)
    movel(p[x_c + -0.024354, y_c + -0.123714, z_c, rx, ry, rz], a, v)
    movel(p[x_c + -0.024683, y_c + -0.123735, z_c, rx, ry, rz], a, v)
    movel(p[x_c + -0.025005, y_c + -0.123758, z_c, rx, ry, rz], a, v)
    movel(p[x_c + -0.025318, y_c + -0.123782, z_c, rx, ry, rz], a, v)
    movel(p[x_c + -0.025624, y_c + -0.123809, z_c, rx, ry, rz], a, v)
    movel(p[x_c + -0.025921, y_c + -0.123838, z_c, rx, ry, rz], a, v)
    movel(p[x_c + -0.026210, y_c + -0.123868, z_c, rx, ry, rz], a, v)
    movel(p[x_c + -0.026491, y_c + -0.123900, z_c, rx, ry, rz], a, v)
    movel(p[x_c + -0.026763, y_c + -0.123935, z_c, rx, ry, rz], a, v)
    movel(p[x_c + -0.027026, y_c + -0.123970, z_c, rx, ry, rz], a, v)
    movel(p[x_c + -0.027280, y_c + -0.124008, z_c, rx, ry, rz], a, v)
    movel(p[x_c + -0.027526, y_c + -0.124048, z_c, rx, ry, rz], a, v)
    movel(p[x_c + -0.027761, y_c + -0.124090, z_c, rx, ry, rz], a, v)
    movel(p[x_c + -0.027987, y_c + -0.124133, z_c, rx, ry, rz], a, v)
    movel(p[x_c + -0.028204, y_c + -0.124178, z_c, rx, ry, rz], a, v)
    movel(p[x_c + -0.028411, y_c + -0.124225, z_c, rx, ry, rz], a, v)
    movel(p[x_c + -0.028607, y_c + -0.124274, z_c, rx, ry, rz], a, v)
    movel(p[x_c + -0.028794, y_c + -0.124325, z_c, rx, ry, rz], a, v)
    movel(p[x_c + -0.028794, y_c + -0.124325, z_c, rx, ry, rz], a, v)
    movel(p[x_c + -0.028807, y_c + -0.124329, z_c, rx, ry, rz], a, v)
    movel(p[x_c + -0.028820, y_c + -0.124332, z_c, rx, ry, rz], a, v)
    movel(p[x_c + -0.028833, y_c + -0.124335, z_c, rx, ry, rz], a, v)
    movel(p[x_c + -0.028846, y_c + -0.124338, z_c, rx, ry, rz], a, v)
    movel(p[x_c + -0.028858, y_c + -0.124341, z_c, rx, ry, rz], a, v)
    movel(p[x_c + -0.028871, y_c + -0.124344, z_c, rx, ry, rz], a, v)
    movel(p[x_c + -0.028883, y_c + -0.124346, z_c, rx, ry, rz], a, v)
    movel(p[x_c + -0.028895, y_c + -0.124348, z_c, rx, ry, rz], a, v)
    movel(p[x_c + -0.028907, y_c + -0.124350, z_c, rx, ry, rz], a, v)
    movel(p[x_c + -0.028919, y_c + -0.124351, z_c, rx, ry, rz], a, v)
    movel(p[x_c + -0.028931, y_c + -0.124353, z_c, rx, ry, rz], a, v)
    movel(p[x_c + -0.028942, y_c + -0.124354, z_c, rx, ry, rz], a, v)
    movel(p[x_c + -0.028954, y_c + -0.124354, z_c, rx, ry, rz], a, v)
    movel(p[x_c + -0.028965, y_c + -0.124355, z_c, rx, ry, rz], a, v)
    movel(p[x_c + -0.028976, y_c + -0.124355, z_c, rx, ry, rz], a, v)
    movel(p[x_c + -0.028987, y_c + -0.124356, z_c, rx, ry, rz], a, v)
    movel(p[x_c + -0.028997, y_c + -0.124356, z_c, rx, ry, rz], a, v)
    movel(p[x_c + -0.029008, y_c + -0.124355, z_c, rx, ry, rz], a, v)
    movel(p[x_c + -0.029018, y_c + -0.124355, z_c, rx, ry, rz], a, v)
    movel(p[x_c + -0.029028, y_c + -0.124354, z_c, rx, ry, rz], a, v)
    movel(p[x_c + -0.029038, y_c + -0.124353, z_c, rx, ry, rz], a, v)
    movel(p[x_c + -0.029047, y_c + -0.124352, z_c, rx, ry, rz], a, v)
    movel(p[x_c + -0.029056, y_c + -0.124351, z_c, rx, ry, rz], a, v)
    movel(p[x_c + -0.029065, y_c + -0.124349, z_c, rx, ry, rz], a, v)
    movel(p[x_c + -0.029074, y_c + -0.124347, z_c, rx, ry, rz], a, v)
    movel(p[x_c + -0.029082, y_c + -0.124345, z_c, rx, ry, rz], a, v)
    movel(p[x_c + -0.029090, y_c + -0.124343, z_c, rx, ry, rz], a, v)
    movel(p[x_c + -0.029098, y_c + -0.124341, z_c, rx, ry, rz], a, v)
    movel(p[x_c + -0.029106, y_c + -0.124338, z_c, rx, ry, rz], a, v)
    movel(p[x_c + -0.029113, y_c + -0.124335, z_c, rx, ry, rz], a, v)
    movel(p[x_c + -0.029120, y_c + -0.124332, z_c, rx, ry, rz], a, v)
    movel(p[x_c + -0.029126, y_c + -0.124329, z_c, rx, ry, rz], a, v)
    movel(p[x_c + -0.029133, y_c + -0.124326, z_c, rx, ry, rz], a, v)
    movel(p[x_c + -0.029139, y_c + -0.124322, z_c, rx, ry, rz], a, v)
    movel(p[x_c + -0.029144, y_c + -0.124318, z_c, rx, ry, rz], a, v)
    movel(p[x_c + -0.029150, y_c + -0.124314, z_c, rx, ry, rz], a, v)
    movel(p[x_c + -0.029155, y_c + -0.124310, z_c, rx, ry, rz], a, v)
    movel(p[x_c + -0.029159, y_c + -0.124306, z_c, rx, ry, rz], a, v)
    movel(p[x_c + -0.029163, y_c + -0.124301, z_c, rx, ry, rz], a, v)
    movel(p[x_c + -0.029167, y_c + -0.124296, z_c, rx, ry, rz], a, v)
    movel(p[x_c + -0.029171, y_c + -0.124291, z_c, rx, ry, rz], a, v)
    movel(p[x_c + -0.029174, y_c + -0.124286, z_c, rx, ry, rz], a, v)
    movel(p[x_c + -0.029177, y_c + -0.124281, z_c, rx, ry, rz], a, v)
    movel(p[x_c + -0.029179, y_c + -0.124276, z_c, rx, ry, rz], a, v)
    movel(p[x_c + -0.029181, y_c + -0.124270, z_c, rx, ry, rz], a, v)
    movel(p[x_c + -0.029182, y_c + -0.124264, z_c, rx, ry, rz], a, v)
    movel(p[x_c + -0.029183, y_c + -0.124258, z_c, rx, ry, rz], a, v)
    movel(p[x_c + -0.029184, y_c + -0.124252, z_c, rx, ry, rz], a, v)
    movel(p[x_c + -0.029184, y_c + -0.124246, z_c, rx, ry, rz], a, v)
    movel(p[x_c + -0.029184, y_c + -0.124246, z_c, rx, ry, rz], a, v)
    movel(p[x_c + -0.029184, y_c + -0.124246, z_c, rx, ry, rz], a, v)
    movel(p[x_c + -0.029184, y_c + -0.124246, z_c, rx, ry, rz], a, v)
    movel(p[x_c + -0.029184, y_c + -0.124246, z_c, rx, ry, rz], a, v)
    movel(p[x_c + -0.029184, y_c + -0.124246, z_c, rx, ry, rz], a, v)
    movel(p[x_c + -0.029184, y_c + -0.124246, z_c, rx, ry, rz], a, v)
    movel(p[x_c + -0.029184, y_c + -0.124246, z_c, rx, ry, rz], a, v)
    movel(p[x_c + -0.029184, y_c + -0.124246, z_c, rx, ry, rz], a, v)
    movel(p[x_c + -0.029184, y_c + -0.124246, z_c, rx, ry, rz], a, v)
    movel(p[x_c + -0.029184, y_c + -0.124246, z_c, rx, ry, rz], a, v)
    movel(p[x_c + 0.021283, y_c + -0.115699, z_c, rx, ry, rz], a, v)
    movel(p[x_c + 0.021283, y_c + -0.115699, z_c, rx, ry, rz], a, v)
    movel(p[x_c + 0.021283, y_c + -0.115699, z_c, rx, ry, rz], a, v)
    movel(p[x_c + 0.021283, y_c + -0.115699, z_c, rx, ry, rz], a, v)
    movel(p[x_c + 0.021283, y_c + -0.115699, z_c, rx, ry, rz], a, v)
    movel(p[x_c + 0.021283, y_c + -0.115699, z_c, rx, ry, rz], a, v)
    movel(p[x_c + 0.021283, y_c + -0.115699, z_c, rx, ry, rz], a, v)
    movel(p[x_c + 0.021283, y_c + -0.115699, z_c, rx, ry, rz], a, v)
    movel(p[x_c + 0.021283, y_c + -0.115699, z_c, rx, ry, rz], a, v)
    movel(p[x_c + 0.021283, y_c + -0.115699, z_c, rx, ry, rz], a, v)
    movel(p[x_c + 0.021283, y_c + -0.115699, z_c, rx, ry, rz], a, v)
    movel(p[x_c + 0.021391, y_c + -0.115668, z_c, rx, ry, rz], a, v)
    movel(p[x_c + 0.021496, y_c + -0.115633, z_c, rx, ry, rz], a, v)
    movel(p[x_c + 0.021599, y_c + -0.115596, z_c, rx, ry, rz], a, v)
    movel(p[x_c + 0.021699, y_c + -0.115556, z_c, rx, ry, rz], a, v)
    movel(p[x_c + 0.021796, y_c + -0.115513, z_c, rx, ry, rz], a, v)
    movel(p[x_c + 0.021890, y_c + -0.115466, z_c, rx, ry, rz], a, v)
    movel(p[x_c + 0.021982, y_c + -0.115417, z_c, rx, ry, rz], a, v)
    movel(p[x_c + 0.022072, y_c + -0.115365, z_c, rx, ry, rz], a, v)
    movel(p[x_c + 0.022158, y_c + -0.115310, z_c, rx, ry, rz], a, v)
    movel(p[x_c + 0.022243, y_c + -0.115251, z_c, rx, ry, rz], a, v)
    movel(p[x_c + 0.022325, y_c + -0.115189, z_c, rx, ry, rz], a, v)
    movel(p[x_c + 0.022404, y_c + -0.115123, z_c, rx, ry, rz], a, v)
    movel(p[x_c + 0.022481, y_c + -0.115054, z_c, rx, ry, rz], a, v)
    movel(p[x_c + 0.022555, y_c + -0.114982, z_c, rx, ry, rz], a, v)
    movel(p[x_c + 0.022627, y_c + -0.114906, z_c, rx, ry, rz], a, v)
    movel(p[x_c + 0.022697, y_c + -0.114826, z_c, rx, ry, rz], a, v)
    movel(p[x_c + 0.022764, y_c + -0.114743, z_c, rx, ry, rz], a, v)
    movel(p[x_c + 0.022829, y_c + -0.114656, z_c, rx, ry, rz], a, v)
    movel(p[x_c + 0.022892, y_c + -0.114564, z_c, rx, ry, rz], a, v)
    movel(p[x_c + 0.022953, y_c + -0.114469, z_c, rx, ry, rz], a, v)
    movel(p[x_c + 0.023011, y_c + -0.114370, z_c, rx, ry, rz], a, v)
    movel(p[x_c + 0.023067, y_c + -0.114267, z_c, rx, ry, rz], a, v)
    movel(p[x_c + 0.023121, y_c + -0.114160, z_c, rx, ry, rz], a, v)
    movel(p[x_c + 0.023173, y_c + -0.114049, z_c, rx, ry, rz], a, v)
    movel(p[x_c + 0.023223, y_c + -0.113933, z_c, rx, ry, rz], a, v)
    movel(p[x_c + 0.023271, y_c + -0.113813, z_c, rx, ry, rz], a, v)
    movel(p[x_c + 0.023317, y_c + -0.113688, z_c, rx, ry, rz], a, v)
    movel(p[x_c + 0.023360, y_c + -0.113559, z_c, rx, ry, rz], a, v)
    movel(p[x_c + 0.023402, y_c + -0.113426, z_c, rx, ry, rz], a, v)
    movel(p[x_c + 0.023442, y_c + -0.113288, z_c, rx, ry, rz], a, v)
    movel(p[x_c + 0.023480, y_c + -0.113145, z_c, rx, ry, rz], a, v)
    movel(p[x_c + 0.023516, y_c + -0.112998, z_c, rx, ry, rz], a, v)
    movel(p[x_c + 0.023550, y_c + -0.112845, z_c, rx, ry, rz], a, v)
    movel(p[x_c + 0.023582, y_c + -0.112688, z_c, rx, ry, rz], a, v)
    movel(p[x_c + 0.023613, y_c + -0.112526, z_c, rx, ry, rz], a, v)
    movel(p[x_c + 0.023642, y_c + -0.112359, z_c, rx, ry, rz], a, v)
    movel(p[x_c + 0.023669, y_c + -0.112187, z_c, rx, ry, rz], a, v)
    movel(p[x_c + 0.023694, y_c + -0.112009, z_c, rx, ry, rz], a, v)
    movel(p[x_c + 0.023717, y_c + -0.111827, z_c, rx, ry, rz], a, v)
    movel(p[x_c + 0.023739, y_c + -0.111639, z_c, rx, ry, rz], a, v)
    movel(p[x_c + 0.023760, y_c + -0.111446, z_c, rx, ry, rz], a, v)
    movel(p[x_c + 0.023778, y_c + -0.111247, z_c, rx, ry, rz], a, v)
    movel(p[x_c + 0.023795, y_c + -0.111043, z_c, rx, ry, rz], a, v)
    movel(p[x_c + 0.023811, y_c + -0.110834, z_c, rx, ry, rz], a, v)
    movel(p[x_c + 0.023825, y_c + -0.110619, z_c, rx, ry, rz], a, v)
    movel(p[x_c + 0.023838, y_c + -0.110398, z_c, rx, ry, rz], a, v)
    movel(p[x_c + 0.023849, y_c + -0.110171, z_c, rx, ry, rz], a, v)
    movel(p[x_c + 0.023858, y_c + -0.109939, z_c, rx, ry, rz], a, v)
    movel(p[x_c + 0.023867, y_c + -0.109700, z_c, rx, ry, rz], a, v)
    movel(p[x_c + 0.023867, y_c + -0.109700, z_c, rx, ry, rz], a, v)
    movel(p[x_c + 0.023953, y_c + -0.106938, z_c, rx, ry, rz], a, v)
    movel(p[x_c + 0.023953, y_c + -0.106938, z_c, rx, ry, rz], a, v)
    movel(p[x_c + 0.025280, y_c + -0.105289, z_c, rx, ry, rz], a, v)
    movel(p[x_c + 0.025280, y_c + -0.105289, z_c, rx, ry, rz], a, v)
    movel(p[x_c + 0.025380, y_c + -0.105163, z_c, rx, ry, rz], a, v)
    movel(p[x_c + 0.025480, y_c + -0.105035, z_c, rx, ry, rz], a, v)
    movel(p[x_c + 0.025579, y_c + -0.104904, z_c, rx, ry, rz], a, v)
    movel(p[x_c + 0.025679, y_c + -0.104770, z_c, rx, ry, rz], a, v)
    movel(p[x_c + 0.025777, y_c + -0.104635, z_c, rx, ry, rz], a, v)
    movel(p[x_c + 0.025876, y_c + -0.104496, z_c, rx, ry, rz], a, v)
    movel(p[x_c + 0.025974, y_c + -0.104356, z_c, rx, ry, rz], a, v)
    movel(p[x_c + 0.026072, y_c + -0.104213, z_c, rx, ry, rz], a, v)
    movel(p[x_c + 0.026169, y_c + -0.104069, z_c, rx, ry, rz], a, v)
    movel(p[x_c + 0.026265, y_c + -0.103922, z_c, rx, ry, rz], a, v)
    movel(p[x_c + 0.026361, y_c + -0.103774, z_c, rx, ry, rz], a, v)
    movel(p[x_c + 0.026457, y_c + -0.103624, z_c, rx, ry, rz], a, v)
    movel(p[x_c + 0.026551, y_c + -0.103472, z_c, rx, ry, rz], a, v)
    movel(p[x_c + 0.026645, y_c + -0.103319, z_c, rx, ry, rz], a, v)
    movel(p[x_c + 0.026738, y_c + -0.103164, z_c, rx, ry, rz], a, v)
    movel(p[x_c + 0.026830, y_c + -0.103008, z_c, rx, ry, rz], a, v)
    movel(p[x_c + 0.026922, y_c + -0.102850, z_c, rx, ry, rz], a, v)
    movel(p[x_c + 0.027012, y_c + -0.102692, z_c, rx, ry, rz], a, v)
    movel(p[x_c + 0.027101, y_c + -0.102532, z_c, rx, ry, rz], a, v)
    movel(p[x_c + 0.027190, y_c + -0.102372, z_c, rx, ry, rz], a, v)
    movel(p[x_c + 0.027277, y_c + -0.102210, z_c, rx, ry, rz], a, v)
    movel(p[x_c + 0.027363, y_c + -0.102048, z_c, rx, ry, rz], a, v)
    movel(p[x_c + 0.027448, y_c + -0.101885, z_c, rx, ry, rz], a, v)
    movel(p[x_c + 0.027531, y_c + -0.101721, z_c, rx, ry, rz], a, v)
    movel(p[x_c + 0.027614, y_c + -0.101557, z_c, rx, ry, rz], a, v)
    movel(p[x_c + 0.027695, y_c + -0.101393, z_c, rx, ry, rz], a, v)
    movel(p[x_c + 0.027774, y_c + -0.101228, z_c, rx, ry, rz], a, v)
    movel(p[x_c + 0.027852, y_c + -0.101064, z_c, rx, ry, rz], a, v)
    movel(p[x_c + 0.027929, y_c + -0.100899, z_c, rx, ry, rz], a, v)
    movel(p[x_c + 0.028004, y_c + -0.100734, z_c, rx, ry, rz], a, v)
    movel(p[x_c + 0.028078, y_c + -0.100569, z_c, rx, ry, rz], a, v)
    movel(p[x_c + 0.028150, y_c + -0.100404, z_c, rx, ry, rz], a, v)
    movel(p[x_c + 0.028220, y_c + -0.100240, z_c, rx, ry, rz], a, v)
    movel(p[x_c + 0.028288, y_c + -0.100076, z_c, rx, ry, rz], a, v)
    movel(p[x_c + 0.028355, y_c + -0.099912, z_c, rx, ry, rz], a, v)
    movel(p[x_c + 0.028420, y_c + -0.099749, z_c, rx, ry, rz], a, v)
    movel(p[x_c + 0.028483, y_c + -0.099587, z_c, rx, ry, rz], a, v)
    movel(p[x_c + 0.028544, y_c + -0.099426, z_c, rx, ry, rz], a, v)
    movel(p[x_c + 0.028603, y_c + -0.099265, z_c, rx, ry, rz], a, v)
    movel(p[x_c + 0.028660, y_c + -0.099106, z_c, rx, ry, rz], a, v)
    movel(p[x_c + 0.028715, y_c + -0.098947, z_c, rx, ry, rz], a, v)
    movel(p[x_c + 0.028768, y_c + -0.098790, z_c, rx, ry, rz], a, v)
    movel(p[x_c + 0.028819, y_c + -0.098634, z_c, rx, ry, rz], a, v)
    movel(p[x_c + 0.028867, y_c + -0.098479, z_c, rx, ry, rz], a, v)
    movel(p[x_c + 0.028913, y_c + -0.098326, z_c, rx, ry, rz], a, v)
    movel(p[x_c + 0.028957, y_c + -0.098174, z_c, rx, ry, rz], a, v)
    movel(p[x_c + 0.028999, y_c + -0.098024, z_c, rx, ry, rz], a, v)
    movel(p[x_c + 0.029038, y_c + -0.097876, z_c, rx, ry, rz], a, v)
    movel(p[x_c + 0.029075, y_c + -0.097729, z_c, rx, ry, rz], a, v)
    movel(p[x_c + 0.029075, y_c + -0.097729, z_c, rx, ry, rz], a, v)
    movel(p[x_c + 0.029101, y_c + -0.097619, z_c, rx, ry, rz], a, v)
    movel(p[x_c + 0.029127, y_c + -0.097503, z_c, rx, ry, rz], a, v)
    movel(p[x_c + 0.029154, y_c + -0.097381, z_c, rx, ry, rz], a, v)
    movel(p[x_c + 0.029180, y_c + -0.097254, z_c, rx, ry, rz], a, v)
    movel(p[x_c + 0.029206, y_c + -0.097121, z_c, rx, ry, rz], a, v)
    movel(p[x_c + 0.029233, y_c + -0.096984, z_c, rx, ry, rz], a, v)
    movel(p[x_c + 0.029259, y_c + -0.096843, z_c, rx, ry, rz], a, v)
    movel(p[x_c + 0.029285, y_c + -0.096696, z_c, rx, ry, rz], a, v)
    movel(p[x_c + 0.029311, y_c + -0.096546, z_c, rx, ry, rz], a, v)
    movel(p[x_c + 0.029337, y_c + -0.096392, z_c, rx, ry, rz], a, v)
    movel(p[x_c + 0.029363, y_c + -0.096234, z_c, rx, ry, rz], a, v)
    movel(p[x_c + 0.029389, y_c + -0.096073, z_c, rx, ry, rz], a, v)
    movel(p[x_c + 0.029414, y_c + -0.095908, z_c, rx, ry, rz], a, v)
    movel(p[x_c + 0.029439, y_c + -0.095741, z_c, rx, ry, rz], a, v)
    movel(p[x_c + 0.029464, y_c + -0.095570, z_c, rx, ry, rz], a, v)
    movel(p[x_c + 0.029489, y_c + -0.095397, z_c, rx, ry, rz], a, v)
    movel(p[x_c + 0.029513, y_c + -0.095222, z_c, rx, ry, rz], a, v)
    movel(p[x_c + 0.029537, y_c + -0.095045, z_c, rx, ry, rz], a, v)
    movel(p[x_c + 0.029561, y_c + -0.094866, z_c, rx, ry, rz], a, v)
    movel(p[x_c + 0.029584, y_c + -0.094685, z_c, rx, ry, rz], a, v)
    movel(p[x_c + 0.029607, y_c + -0.094502, z_c, rx, ry, rz], a, v)
    movel(p[x_c + 0.029629, y_c + -0.094319, z_c, rx, ry, rz], a, v)
    movel(p[x_c + 0.029651, y_c + -0.094135, z_c, rx, ry, rz], a, v)
    movel(p[x_c + 0.029673, y_c + -0.093950, z_c, rx, ry, rz], a, v)
    movel(p[x_c + 0.029694, y_c + -0.093764, z_c, rx, ry, rz], a, v)
    movel(p[x_c + 0.029714, y_c + -0.093578, z_c, rx, ry, rz], a, v)
    movel(p[x_c + 0.029734, y_c + -0.093392, z_c, rx, ry, rz], a, v)
    movel(p[x_c + 0.029753, y_c + -0.093207, z_c, rx, ry, rz], a, v)
    movel(p[x_c + 0.029771, y_c + -0.093021, z_c, rx, ry, rz], a, v)
    movel(p[x_c + 0.029789, y_c + -0.092837, z_c, rx, ry, rz], a, v)
    movel(p[x_c + 0.029807, y_c + -0.092653, z_c, rx, ry, rz], a, v)
    movel(p[x_c + 0.029823, y_c + -0.092470, z_c, rx, ry, rz], a, v)
    movel(p[x_c + 0.029839, y_c + -0.092289, z_c, rx, ry, rz], a, v)
    movel(p[x_c + 0.029854, y_c + -0.092110, z_c, rx, ry, rz], a, v)
    movel(p[x_c + 0.029868, y_c + -0.091932, z_c, rx, ry, rz], a, v)
    movel(p[x_c + 0.029882, y_c + -0.091756, z_c, rx, ry, rz], a, v)
    movel(p[x_c + 0.029894, y_c + -0.091582, z_c, rx, ry, rz], a, v)
    movel(p[x_c + 0.029906, y_c + -0.091411, z_c, rx, ry, rz], a, v)
    movel(p[x_c + 0.029917, y_c + -0.091243, z_c, rx, ry, rz], a, v)
    movel(p[x_c + 0.029927, y_c + -0.091077, z_c, rx, ry, rz], a, v)
    movel(p[x_c + 0.029936, y_c + -0.090915, z_c, rx, ry, rz], a, v)
    movel(p[x_c + 0.029944, y_c + -0.090756, z_c, rx, ry, rz], a, v)
    movel(p[x_c + 0.029951, y_c + -0.090601, z_c, rx, ry, rz], a, v)
    movel(p[x_c + 0.029957, y_c + -0.090450, z_c, rx, ry, rz], a, v)
    movel(p[x_c + 0.029963, y_c + -0.090303, z_c, rx, ry, rz], a, v)
    movel(p[x_c + 0.029967, y_c + -0.090160, z_c, rx, ry, rz], a, v)
    movel(p[x_c + 0.029969, y_c + -0.090021, z_c, rx, ry, rz], a, v)
    movel(p[x_c + 0.029971, y_c + -0.089888, z_c, rx, ry, rz], a, v)
    movel(p[x_c + 0.029972, y_c + -0.089759, z_c, rx, ry, rz], a, v)
    movel(p[x_c + 0.029972, y_c + -0.089759, z_c, rx, ry, rz], a, v)
    movel(p[x_c + 0.029972, y_c + -0.089706, z_c, rx, ry, rz], a, v)
    movel(p[x_c + 0.029973, y_c + -0.089654, z_c, rx, ry, rz], a, v)
    movel(p[x_c + 0.029974, y_c + -0.089602, z_c, rx, ry, rz], a, v)
    movel(p[x_c + 0.029975, y_c + -0.089552, z_c, rx, ry, rz], a, v)
    movel(p[x_c + 0.029978, y_c + -0.089503, z_c, rx, ry, rz], a, v)
    movel(p[x_c + 0.029980, y_c + -0.089455, z_c, rx, ry, rz], a, v)
    movel(p[x_c + 0.029983, y_c + -0.089407, z_c, rx, ry, rz], a, v)
    movel(p[x_c + 0.029987, y_c + -0.089360, z_c, rx, ry, rz], a, v)
    movel(p[x_c + 0.029992, y_c + -0.089314, z_c, rx, ry, rz], a, v)
    movel(p[x_c + 0.029997, y_c + -0.089269, z_c, rx, ry, rz], a, v)
    movel(p[x_c + 0.030002, y_c + -0.089224, z_c, rx, ry, rz], a, v)
    movel(p[x_c + 0.030009, y_c + -0.089179, z_c, rx, ry, rz], a, v)
    movel(p[x_c + 0.030016, y_c + -0.089135, z_c, rx, ry, rz], a, v)
    movel(p[x_c + 0.030024, y_c + -0.089091, z_c, rx, ry, rz], a, v)
    movel(p[x_c + 0.030032, y_c + -0.089048, z_c, rx, ry, rz], a, v)
    movel(p[x_c + 0.030042, y_c + -0.089005, z_c, rx, ry, rz], a, v)
    movel(p[x_c + 0.030052, y_c + -0.088962, z_c, rx, ry, rz], a, v)
    movel(p[x_c + 0.030063, y_c + -0.088919, z_c, rx, ry, rz], a, v)
    movel(p[x_c + 0.030076, y_c + -0.088876, z_c, rx, ry, rz], a, v)
    movel(p[x_c + 0.030089, y_c + -0.088832, z_c, rx, ry, rz], a, v)
    movel(p[x_c + 0.030102, y_c + -0.088789, z_c, rx, ry, rz], a, v)
    movel(p[x_c + 0.030117, y_c + -0.088746, z_c, rx, ry, rz], a, v)
    movel(p[x_c + 0.030133, y_c + -0.088702, z_c, rx, ry, rz], a, v)
    movel(p[x_c + 0.030150, y_c + -0.088658, z_c, rx, ry, rz], a, v)
    movel(p[x_c + 0.030168, y_c + -0.088614, z_c, rx, ry, rz], a, v)
    movel(p[x_c + 0.030187, y_c + -0.088569, z_c, rx, ry, rz], a, v)
    movel(p[x_c + 0.030207, y_c + -0.088524, z_c, rx, ry, rz], a, v)
    movel(p[x_c + 0.030229, y_c + -0.088478, z_c, rx, ry, rz], a, v)
    movel(p[x_c + 0.030251, y_c + -0.088432, z_c, rx, ry, rz], a, v)
    movel(p[x_c + 0.030275, y_c + -0.088385, z_c, rx, ry, rz], a, v)
    movel(p[x_c + 0.030300, y_c + -0.088336, z_c, rx, ry, rz], a, v)
    movel(p[x_c + 0.030326, y_c + -0.088288, z_c, rx, ry, rz], a, v)
    movel(p[x_c + 0.030353, y_c + -0.088238, z_c, rx, ry, rz], a, v)
    movel(p[x_c + 0.030382, y_c + -0.088187, z_c, rx, ry, rz], a, v)
    movel(p[x_c + 0.030412, y_c + -0.088135, z_c, rx, ry, rz], a, v)
    movel(p[x_c + 0.030443, y_c + -0.088082, z_c, rx, ry, rz], a, v)
    movel(p[x_c + 0.030476, y_c + -0.088028, z_c, rx, ry, rz], a, v)
    movel(p[x_c + 0.030510, y_c + -0.087973, z_c, rx, ry, rz], a, v)
    movel(p[x_c + 0.030545, y_c + -0.087916, z_c, rx, ry, rz], a, v)
    movel(p[x_c + 0.030582, y_c + -0.087858, z_c, rx, ry, rz], a, v)
    movel(p[x_c + 0.030621, y_c + -0.087798, z_c, rx, ry, rz], a, v)
    movel(p[x_c + 0.030661, y_c + -0.087737, z_c, rx, ry, rz], a, v)
    movel(p[x_c + 0.030702, y_c + -0.087675, z_c, rx, ry, rz], a, v)
    movel(p[x_c + 0.030745, y_c + -0.087610, z_c, rx, ry, rz], a, v)
    movel(p[x_c + 0.030790, y_c + -0.087544, z_c, rx, ry, rz], a, v)
    movel(p[x_c + 0.030836, y_c + -0.087477, z_c, rx, ry, rz], a, v)
    movel(p[x_c + 0.030884, y_c + -0.087407, z_c, rx, ry, rz], a, v)
    movel(p[x_c + 0.030934, y_c + -0.087335, z_c, rx, ry, rz], a, v)
    movel(p[x_c + 0.030985, y_c + -0.087262, z_c, rx, ry, rz], a, v)
    movel(p[x_c + 0.030985, y_c + -0.087262, z_c, rx, ry, rz], a, v)
    movel(p[x_c + 0.031080, y_c + -0.087124, z_c, rx, ry, rz], a, v)
    movel(p[x_c + 0.031175, y_c + -0.086983, z_c, rx, ry, rz], a, v)
    movel(p[x_c + 0.031269, y_c + -0.086838, z_c, rx, ry, rz], a, v)
    movel(p[x_c + 0.031363, y_c + -0.086691, z_c, rx, ry, rz], a, v)
    movel(p[x_c + 0.031457, y_c + -0.086541, z_c, rx, ry, rz], a, v)
    movel(p[x_c + 0.031550, y_c + -0.086389, z_c, rx, ry, rz], a, v)
    movel(p[x_c + 0.031642, y_c + -0.086234, z_c, rx, ry, rz], a, v)
    movel(p[x_c + 0.031733, y_c + -0.086076, z_c, rx, ry, rz], a, v)
    movel(p[x_c + 0.031824, y_c + -0.085917, z_c, rx, ry, rz], a, v)
    movel(p[x_c + 0.031913, y_c + -0.085756, z_c, rx, ry, rz], a, v)
    movel(p[x_c + 0.032002, y_c + -0.085593, z_c, rx, ry, rz], a, v)
    movel(p[x_c + 0.032090, y_c + -0.085429, z_c, rx, ry, rz], a, v)
    movel(p[x_c + 0.032176, y_c + -0.085263, z_c, rx, ry, rz], a, v)
    movel(p[x_c + 0.032262, y_c + -0.085097, z_c, rx, ry, rz], a, v)
    movel(p[x_c + 0.032346, y_c + -0.084929, z_c, rx, ry, rz], a, v)
    movel(p[x_c + 0.032429, y_c + -0.084760, z_c, rx, ry, rz], a, v)
    movel(p[x_c + 0.032510, y_c + -0.084590, z_c, rx, ry, rz], a, v)
    movel(p[x_c + 0.032590, y_c + -0.084420, z_c, rx, ry, rz], a, v)
    movel(p[x_c + 0.032669, y_c + -0.084250, z_c, rx, ry, rz], a, v)
    movel(p[x_c + 0.032746, y_c + -0.084079, z_c, rx, ry, rz], a, v)
    movel(p[x_c + 0.032822, y_c + -0.083909, z_c, rx, ry, rz], a, v)
    movel(p[x_c + 0.032895, y_c + -0.083738, z_c, rx, ry, rz], a, v)
    movel(p[x_c + 0.032967, y_c + -0.083568, z_c, rx, ry, rz], a, v)
    movel(p[x_c + 0.033037, y_c + -0.083399, z_c, rx, ry, rz], a, v)
    movel(p[x_c + 0.033105, y_c + -0.083230, z_c, rx, ry, rz], a, v)
    movel(p[x_c + 0.033172, y_c + -0.083061, z_c, rx, ry, rz], a, v)
    movel(p[x_c + 0.033236, y_c + -0.082894, z_c, rx, ry, rz], a, v)
    movel(p[x_c + 0.033298, y_c + -0.082728, z_c, rx, ry, rz], a, v)
    movel(p[x_c + 0.033358, y_c + -0.082564, z_c, rx, ry, rz], a, v)
    movel(p[x_c + 0.033415, y_c + -0.082401, z_c, rx, ry, rz], a, v)
    movel(p[x_c + 0.033471, y_c + -0.082239, z_c, rx, ry, rz], a, v)
    movel(p[x_c + 0.033524, y_c + -0.082080, z_c, rx, ry, rz], a, v)
    movel(p[x_c + 0.033574, y_c + -0.081922, z_c, rx, ry, rz], a, v)
    movel(p[x_c + 0.033622, y_c + -0.081767, z_c, rx, ry, rz], a, v)
    movel(p[x_c + 0.033667, y_c + -0.081614, z_c, rx, ry, rz], a, v)
    movel(p[x_c + 0.033710, y_c + -0.081463, z_c, rx, ry, rz], a, v)
    movel(p[x_c + 0.033750, y_c + -0.081315, z_c, rx, ry, rz], a, v)
    movel(p[x_c + 0.033787, y_c + -0.081170, z_c, rx, ry, rz], a, v)
    movel(p[x_c + 0.033821, y_c + -0.081028, z_c, rx, ry, rz], a, v)
    movel(p[x_c + 0.033852, y_c + -0.080890, z_c, rx, ry, rz], a, v)
    movel(p[x_c + 0.033881, y_c + -0.080754, z_c, rx, ry, rz], a, v)
    movel(p[x_c + 0.033906, y_c + -0.080622, z_c, rx, ry, rz], a, v)
    movel(p[x_c + 0.033928, y_c + -0.080494, z_c, rx, ry, rz], a, v)
    movel(p[x_c + 0.033947, y_c + -0.080370, z_c, rx, ry, rz], a, v)
    movel(p[x_c + 0.033963, y_c + -0.080250, z_c, rx, ry, rz], a, v)
    movel(p[x_c + 0.033975, y_c + -0.080134, z_c, rx, ry, rz], a, v)
    movel(p[x_c + 0.033984, y_c + -0.080022, z_c, rx, ry, rz], a, v)
    movel(p[x_c + 0.033989, y_c + -0.079915, z_c, rx, ry, rz], a, v)
    movel(p[x_c + 0.033991, y_c + -0.079813, z_c, rx, ry, rz], a, v)
    movel(p[x_c + 0.033991, y_c + -0.079813, z_c, rx, ry, rz], a, v)
    movel(p[x_c + 0.033990, y_c + -0.079797, z_c, rx, ry, rz], a, v)
    movel(p[x_c + 0.033987, y_c + -0.079778, z_c, rx, ry, rz], a, v)
    movel(p[x_c + 0.033982, y_c + -0.079758, z_c, rx, ry, rz], a, v)
    movel(p[x_c + 0.033974, y_c + -0.079736, z_c, rx, ry, rz], a, v)
    movel(p[x_c + 0.033965, y_c + -0.079712, z_c, rx, ry, rz], a, v)
    movel(p[x_c + 0.033954, y_c + -0.079686, z_c, rx, ry, rz], a, v)
    movel(p[x_c + 0.033941, y_c + -0.079659, z_c, rx, ry, rz], a, v)
    movel(p[x_c + 0.033927, y_c + -0.079630, z_c, rx, ry, rz], a, v)
    movel(p[x_c + 0.033910, y_c + -0.079599, z_c, rx, ry, rz], a, v)
    movel(p[x_c + 0.033891, y_c + -0.079567, z_c, rx, ry, rz], a, v)
    movel(p[x_c + 0.033871, y_c + -0.079533, z_c, rx, ry, rz], a, v)
    movel(p[x_c + 0.033849, y_c + -0.079498, z_c, rx, ry, rz], a, v)
    movel(p[x_c + 0.033825, y_c + -0.079461, z_c, rx, ry, rz], a, v)
    movel(p[x_c + 0.033800, y_c + -0.079422, z_c, rx, ry, rz], a, v)
    movel(p[x_c + 0.033772, y_c + -0.079383, z_c, rx, ry, rz], a, v)
    movel(p[x_c + 0.033743, y_c + -0.079341, z_c, rx, ry, rz], a, v)
    movel(p[x_c + 0.033713, y_c + -0.079299, z_c, rx, ry, rz], a, v)
    movel(p[x_c + 0.033680, y_c + -0.079255, z_c, rx, ry, rz], a, v)
    movel(p[x_c + 0.033647, y_c + -0.079209, z_c, rx, ry, rz], a, v)
    movel(p[x_c + 0.033611, y_c + -0.079162, z_c, rx, ry, rz], a, v)
    movel(p[x_c + 0.033574, y_c + -0.079115, z_c, rx, ry, rz], a, v)
    movel(p[x_c + 0.033536, y_c + -0.079065, z_c, rx, ry, rz], a, v)
    movel(p[x_c + 0.033496, y_c + -0.079015, z_c, rx, ry, rz], a, v)
    movel(p[x_c + 0.033454, y_c + -0.078963, z_c, rx, ry, rz], a, v)
    movel(p[x_c + 0.033411, y_c + -0.078911, z_c, rx, ry, rz], a, v)
    movel(p[x_c + 0.033367, y_c + -0.078857, z_c, rx, ry, rz], a, v)
    movel(p[x_c + 0.033321, y_c + -0.078802, z_c, rx, ry, rz], a, v)
    movel(p[x_c + 0.033274, y_c + -0.078746, z_c, rx, ry, rz], a, v)
    movel(p[x_c + 0.033226, y_c + -0.078689, z_c, rx, ry, rz], a, v)
    movel(p[x_c + 0.033176, y_c + -0.078631, z_c, rx, ry, rz], a, v)
    movel(p[x_c + 0.033125, y_c + -0.078573, z_c, rx, ry, rz], a, v)
    movel(p[x_c + 0.033072, y_c + -0.078513, z_c, rx, ry, rz], a, v)
    movel(p[x_c + 0.033019, y_c + -0.078452, z_c, rx, ry, rz], a, v)
    movel(p[x_c + 0.032964, y_c + -0.078391, z_c, rx, ry, rz], a, v)
    movel(p[x_c + 0.032908, y_c + -0.078329, z_c, rx, ry, rz], a, v)
    movel(p[x_c + 0.032851, y_c + -0.078266, z_c, rx, ry, rz], a, v)
    movel(p[x_c + 0.032793, y_c + -0.078202, z_c, rx, ry, rz], a, v)
    movel(p[x_c + 0.032734, y_c + -0.078137, z_c, rx, ry, rz], a, v)
    movel(p[x_c + 0.032673, y_c + -0.078072, z_c, rx, ry, rz], a, v)
    movel(p[x_c + 0.032612, y_c + -0.078006, z_c, rx, ry, rz], a, v)
    movel(p[x_c + 0.032549, y_c + -0.077940, z_c, rx, ry, rz], a, v)
    movel(p[x_c + 0.032486, y_c + -0.077873, z_c, rx, ry, rz], a, v)
    movel(p[x_c + 0.032421, y_c + -0.077805, z_c, rx, ry, rz], a, v)
    movel(p[x_c + 0.032356, y_c + -0.077737, z_c, rx, ry, rz], a, v)
    movel(p[x_c + 0.032290, y_c + -0.077668, z_c, rx, ry, rz], a, v)
    movel(p[x_c + 0.032223, y_c + -0.077599, z_c, rx, ry, rz], a, v)
    movel(p[x_c + 0.032154, y_c + -0.077530, z_c, rx, ry, rz], a, v)
    movel(p[x_c + 0.032086, y_c + -0.077460, z_c, rx, ry, rz], a, v)
    movel(p[x_c + 0.032016, y_c + -0.077390, z_c, rx, ry, rz], a, v)
    movel(p[x_c + 0.032016, y_c + -0.077390, z_c, rx, ry, rz], a, v)
    movel(p[x_c + 0.031691, y_c + -0.077059, z_c, rx, ry, rz], a, v)
    movel(p[x_c + 0.031369, y_c + -0.076722, z_c, rx, ry, rz], a, v)
    movel(p[x_c + 0.031049, y_c + -0.076377, z_c, rx, ry, rz], a, v)
    movel(p[x_c + 0.030731, y_c + -0.076026, z_c, rx, ry, rz], a, v)
    movel(p[x_c + 0.030415, y_c + -0.075669, z_c, rx, ry, rz], a, v)
    movel(p[x_c + 0.030102, y_c + -0.075305, z_c, rx, ry, rz], a, v)
    movel(p[x_c + 0.029791, y_c + -0.074934, z_c, rx, ry, rz], a, v)
    movel(p[x_c + 0.029483, y_c + -0.074557, z_c, rx, ry, rz], a, v)
    movel(p[x_c + 0.029177, y_c + -0.074174, z_c, rx, ry, rz], a, v)
    movel(p[x_c + 0.028874, y_c + -0.073785, z_c, rx, ry, rz], a, v)
    movel(p[x_c + 0.028573, y_c + -0.073389, z_c, rx, ry, rz], a, v)
    movel(p[x_c + 0.028275, y_c + -0.072988, z_c, rx, ry, rz], a, v)
    movel(p[x_c + 0.027980, y_c + -0.072581, z_c, rx, ry, rz], a, v)
    movel(p[x_c + 0.027687, y_c + -0.072168, z_c, rx, ry, rz], a, v)
    movel(p[x_c + 0.027398, y_c + -0.071749, z_c, rx, ry, rz], a, v)
    movel(p[x_c + 0.027111, y_c + -0.071325, z_c, rx, ry, rz], a, v)
    movel(p[x_c + 0.026827, y_c + -0.070895, z_c, rx, ry, rz], a, v)
    movel(p[x_c + 0.026547, y_c + -0.070460, z_c, rx, ry, rz], a, v)
    movel(p[x_c + 0.026269, y_c + -0.070019, z_c, rx, ry, rz], a, v)
    movel(p[x_c + 0.025994, y_c + -0.069574, z_c, rx, ry, rz], a, v)
    movel(p[x_c + 0.025723, y_c + -0.069123, z_c, rx, ry, rz], a, v)
    movel(p[x_c + 0.025454, y_c + -0.068667, z_c, rx, ry, rz], a, v)
    movel(p[x_c + 0.025189, y_c + -0.068206, z_c, rx, ry, rz], a, v)
    movel(p[x_c + 0.024928, y_c + -0.067741, z_c, rx, ry, rz], a, v)
    movel(p[x_c + 0.024669, y_c + -0.067270, z_c, rx, ry, rz], a, v)
    movel(p[x_c + 0.024414, y_c + -0.066795, z_c, rx, ry, rz], a, v)
    movel(p[x_c + 0.024163, y_c + -0.066315, z_c, rx, ry, rz], a, v)
    movel(p[x_c + 0.023914, y_c + -0.065831, z_c, rx, ry, rz], a, v)
    movel(p[x_c + 0.023670, y_c + -0.065343, z_c, rx, ry, rz], a, v)
    movel(p[x_c + 0.023429, y_c + -0.064850, z_c, rx, ry, rz], a, v)
    movel(p[x_c + 0.023192, y_c + -0.064353, z_c, rx, ry, rz], a, v)
    movel(p[x_c + 0.022958, y_c + -0.063852, z_c, rx, ry, rz], a, v)
    movel(p[x_c + 0.022728, y_c + -0.063347, z_c, rx, ry, rz], a, v)
    movel(p[x_c + 0.022502, y_c + -0.062838, z_c, rx, ry, rz], a, v)
    movel(p[x_c + 0.022280, y_c + -0.062325, z_c, rx, ry, rz], a, v)
    movel(p[x_c + 0.022062, y_c + -0.061808, z_c, rx, ry, rz], a, v)
    movel(p[x_c + 0.021848, y_c + -0.061288, z_c, rx, ry, rz], a, v)
    movel(p[x_c + 0.021637, y_c + -0.060764, z_c, rx, ry, rz], a, v)
    movel(p[x_c + 0.021431, y_c + -0.060237, z_c, rx, ry, rz], a, v)
    movel(p[x_c + 0.021229, y_c + -0.059707, z_c, rx, ry, rz], a, v)
    movel(p[x_c + 0.021031, y_c + -0.059173, z_c, rx, ry, rz], a, v)
    movel(p[x_c + 0.020837, y_c + -0.058636, z_c, rx, ry, rz], a, v)
    movel(p[x_c + 0.020648, y_c + -0.058096, z_c, rx, ry, rz], a, v)
    movel(p[x_c + 0.020463, y_c + -0.057553, z_c, rx, ry, rz], a, v)
    movel(p[x_c + 0.020282, y_c + -0.057007, z_c, rx, ry, rz], a, v)
    movel(p[x_c + 0.020106, y_c + -0.056458, z_c, rx, ry, rz], a, v)
    movel(p[x_c + 0.019934, y_c + -0.055907, z_c, rx, ry, rz], a, v)
    movel(p[x_c + 0.019766, y_c + -0.055353, z_c, rx, ry, rz], a, v)
    movel(p[x_c + 0.019604, y_c + -0.054796, z_c, rx, ry, rz], a, v)
    movel(p[x_c + 0.019604, y_c + -0.054796, z_c, rx, ry, rz], a, v)
    movel(p[x_c + 0.019439, y_c + -0.054216, z_c, rx, ry, rz], a, v)
    movel(p[x_c + 0.019279, y_c + -0.053635, z_c, rx, ry, rz], a, v)
    movel(p[x_c + 0.019124, y_c + -0.053053, z_c, rx, ry, rz], a, v)
    movel(p[x_c + 0.018974, y_c + -0.052470, z_c, rx, ry, rz], a, v)
    movel(p[x_c + 0.018828, y_c + -0.051885, z_c, rx, ry, rz], a, v)
    movel(p[x_c + 0.018687, y_c + -0.051298, z_c, rx, ry, rz], a, v)
    movel(p[x_c + 0.018550, y_c + -0.050709, z_c, rx, ry, rz], a, v)
    movel(p[x_c + 0.018418, y_c + -0.050118, z_c, rx, ry, rz], a, v)
    movel(p[x_c + 0.018290, y_c + -0.049523, z_c, rx, ry, rz], a, v)
    movel(p[x_c + 0.018167, y_c + -0.048925, z_c, rx, ry, rz], a, v)
    movel(p[x_c + 0.018049, y_c + -0.048324, z_c, rx, ry, rz], a, v)
    movel(p[x_c + 0.017934, y_c + -0.047718, z_c, rx, ry, rz], a, v)
    movel(p[x_c + 0.017824, y_c + -0.047108, z_c, rx, ry, rz], a, v)
    movel(p[x_c + 0.017719, y_c + -0.046494, z_c, rx, ry, rz], a, v)
    movel(p[x_c + 0.017618, y_c + -0.045874, z_c, rx, ry, rz], a, v)
    movel(p[x_c + 0.017521, y_c + -0.045250, z_c, rx, ry, rz], a, v)
    movel(p[x_c + 0.017428, y_c + -0.044619, z_c, rx, ry, rz], a, v)
    movel(p[x_c + 0.017340, y_c + -0.043983, z_c, rx, ry, rz], a, v)
    movel(p[x_c + 0.017256, y_c + -0.043340, z_c, rx, ry, rz], a, v)
    movel(p[x_c + 0.017176, y_c + -0.042690, z_c, rx, ry, rz], a, v)
    movel(p[x_c + 0.017100, y_c + -0.042034, z_c, rx, ry, rz], a, v)
    movel(p[x_c + 0.017028, y_c + -0.041370, z_c, rx, ry, rz], a, v)
    movel(p[x_c + 0.016961, y_c + -0.040698, z_c, rx, ry, rz], a, v)
    movel(p[x_c + 0.016897, y_c + -0.040018, z_c, rx, ry, rz], a, v)
    movel(p[x_c + 0.016838, y_c + -0.039330, z_c, rx, ry, rz], a, v)
    movel(p[x_c + 0.016782, y_c + -0.038633, z_c, rx, ry, rz], a, v)
    movel(p[x_c + 0.016731, y_c + -0.037927, z_c, rx, ry, rz], a, v)
    movel(p[x_c + 0.016683, y_c + -0.037212, z_c, rx, ry, rz], a, v)
    movel(p[x_c + 0.016640, y_c + -0.036486, z_c, rx, ry, rz], a, v)
    movel(p[x_c + 0.016600, y_c + -0.035751, z_c, rx, ry, rz], a, v)
    movel(p[x_c + 0.016564, y_c + -0.035005, z_c, rx, ry, rz], a, v)
    movel(p[x_c + 0.016532, y_c + -0.034249, z_c, rx, ry, rz], a, v)
    movel(p[x_c + 0.016504, y_c + -0.033481, z_c, rx, ry, rz], a, v)
    movel(p[x_c + 0.016479, y_c + -0.032702, z_c, rx, ry, rz], a, v)
    movel(p[x_c + 0.016459, y_c + -0.031911, z_c, rx, ry, rz], a, v)
    movel(p[x_c + 0.016442, y_c + -0.031108, z_c, rx, ry, rz], a, v)
    movel(p[x_c + 0.016429, y_c + -0.030293, z_c, rx, ry, rz], a, v)
    movel(p[x_c + 0.016419, y_c + -0.029464, z_c, rx, ry, rz], a, v)
    movel(p[x_c + 0.016413, y_c + -0.028623, z_c, rx, ry, rz], a, v)
    movel(p[x_c + 0.016411, y_c + -0.027768, z_c, rx, ry, rz], a, v)
    movel(p[x_c + 0.016412, y_c + -0.026899, z_c, rx, ry, rz], a, v)
    movel(p[x_c + 0.016416, y_c + -0.026016, z_c, rx, ry, rz], a, v)
    movel(p[x_c + 0.016425, y_c + -0.025118, z_c, rx, ry, rz], a, v)
    movel(p[x_c + 0.016436, y_c + -0.024206, z_c, rx, ry, rz], a, v)
    movel(p[x_c + 0.016451, y_c + -0.023278, z_c, rx, ry, rz], a, v)
    movel(p[x_c + 0.016470, y_c + -0.022335, z_c, rx, ry, rz], a, v)
    movel(p[x_c + 0.016492, y_c + -0.021376, z_c, rx, ry, rz], a, v)
    movel(p[x_c + 0.016517, y_c + -0.020401, z_c, rx, ry, rz], a, v)
    movel(p[x_c + 0.016546, y_c + -0.019409, z_c, rx, ry, rz], a, v)
    movel(p[x_c + 0.016546, y_c + -0.019409, z_c, rx, ry, rz], a, v)
    movel(p[x_c + 0.016556, y_c + -0.019099, z_c, rx, ry, rz], a, v)
    movel(p[x_c + 0.016565, y_c + -0.018786, z_c, rx, ry, rz], a, v)
    movel(p[x_c + 0.016575, y_c + -0.018470, z_c, rx, ry, rz], a, v)
    movel(p[x_c + 0.016585, y_c + -0.018153, z_c, rx, ry, rz], a, v)
    movel(p[x_c + 0.016596, y_c + -0.017835, z_c, rx, ry, rz], a, v)
    movel(p[x_c + 0.016607, y_c + -0.017514, z_c, rx, ry, rz], a, v)
    movel(p[x_c + 0.016617, y_c + -0.017193, z_c, rx, ry, rz], a, v)
    movel(p[x_c + 0.016628, y_c + -0.016871, z_c, rx, ry, rz], a, v)
    movel(p[x_c + 0.016640, y_c + -0.016548, z_c, rx, ry, rz], a, v)
    movel(p[x_c + 0.016651, y_c + -0.016224, z_c, rx, ry, rz], a, v)
    movel(p[x_c + 0.016662, y_c + -0.015901, z_c, rx, ry, rz], a, v)
    movel(p[x_c + 0.016674, y_c + -0.015577, z_c, rx, ry, rz], a, v)
    movel(p[x_c + 0.016686, y_c + -0.015254, z_c, rx, ry, rz], a, v)
    movel(p[x_c + 0.016698, y_c + -0.014931, z_c, rx, ry, rz], a, v)
    movel(p[x_c + 0.016710, y_c + -0.014609, z_c, rx, ry, rz], a, v)
    movel(p[x_c + 0.016722, y_c + -0.014288, z_c, rx, ry, rz], a, v)
    movel(p[x_c + 0.016734, y_c + -0.013968, z_c, rx, ry, rz], a, v)
    movel(p[x_c + 0.016746, y_c + -0.013650, z_c, rx, ry, rz], a, v)
    movel(p[x_c + 0.016759, y_c + -0.013333, z_c, rx, ry, rz], a, v)
    movel(p[x_c + 0.016771, y_c + -0.013019, z_c, rx, ry, rz], a, v)
    movel(p[x_c + 0.016784, y_c + -0.012706, z_c, rx, ry, rz], a, v)
    movel(p[x_c + 0.016796, y_c + -0.012396, z_c, rx, ry, rz], a, v)
    movel(p[x_c + 0.016809, y_c + -0.012089, z_c, rx, ry, rz], a, v)
    movel(p[x_c + 0.016822, y_c + -0.011785, z_c, rx, ry, rz], a, v)
    movel(p[x_c + 0.016834, y_c + -0.011484, z_c, rx, ry, rz], a, v)
    movel(p[x_c + 0.016847, y_c + -0.011186, z_c, rx, ry, rz], a, v)
    movel(p[x_c + 0.016859, y_c + -0.010892, z_c, rx, ry, rz], a, v)
    movel(p[x_c + 0.016872, y_c + -0.010602, z_c, rx, ry, rz], a, v)
    movel(p[x_c + 0.016885, y_c + -0.010316, z_c, rx, ry, rz], a, v)
    movel(p[x_c + 0.016897, y_c + -0.010034, z_c, rx, ry, rz], a, v)
    movel(p[x_c + 0.016910, y_c + -0.009758, z_c, rx, ry, rz], a, v)
    movel(p[x_c + 0.016922, y_c + -0.009485, z_c, rx, ry, rz], a, v)
    movel(p[x_c + 0.016934, y_c + -0.009219, z_c, rx, ry, rz], a, v)
    movel(p[x_c + 0.016947, y_c + -0.008957, z_c, rx, ry, rz], a, v)
    movel(p[x_c + 0.016959, y_c + -0.008701, z_c, rx, ry, rz], a, v)
    movel(p[x_c + 0.016971, y_c + -0.008451, z_c, rx, ry, rz], a, v)
    movel(p[x_c + 0.016983, y_c + -0.008207, z_c, rx, ry, rz], a, v)
    movel(p[x_c + 0.016995, y_c + -0.007969, z_c, rx, ry, rz], a, v)
    movel(p[x_c + 0.017007, y_c + -0.007738, z_c, rx, ry, rz], a, v)
    movel(p[x_c + 0.017018, y_c + -0.007514, z_c, rx, ry, rz], a, v)
    movel(p[x_c + 0.017030, y_c + -0.007296, z_c, rx, ry, rz], a, v)
    movel(p[x_c + 0.017041, y_c + -0.007086, z_c, rx, ry, rz], a, v)
    movel(p[x_c + 0.017052, y_c + -0.006884, z_c, rx, ry, rz], a, v)
    movel(p[x_c + 0.017063, y_c + -0.006689, z_c, rx, ry, rz], a, v)
    movel(p[x_c + 0.017074, y_c + -0.006503, z_c, rx, ry, rz], a, v)
    movel(p[x_c + 0.017084, y_c + -0.006325, z_c, rx, ry, rz], a, v)
    movel(p[x_c + 0.017095, y_c + -0.006155, z_c, rx, ry, rz], a, v)
    movel(p[x_c + 0.017105, y_c + -0.005994, z_c, rx, ry, rz], a, v)
    movel(p[x_c + 0.017115, y_c + -0.005842, z_c, rx, ry, rz], a, v)
    movel(p[x_c + 0.017115, y_c + -0.005842, z_c, rx, ry, rz], a, v)
    movel(p[x_c + 0.017125, y_c + -0.005694, z_c, rx, ry, rz], a, v)
    movel(p[x_c + 0.017134, y_c + -0.005546, z_c, rx, ry, rz], a, v)
    movel(p[x_c + 0.017143, y_c + -0.005398, z_c, rx, ry, rz], a, v)
    movel(p[x_c + 0.017152, y_c + -0.005250, z_c, rx, ry, rz], a, v)
    movel(p[x_c + 0.017160, y_c + -0.005103, z_c, rx, ry, rz], a, v)
    movel(p[x_c + 0.017169, y_c + -0.004955, z_c, rx, ry, rz], a, v)
    movel(p[x_c + 0.017177, y_c + -0.004808, z_c, rx, ry, rz], a, v)
    movel(p[x_c + 0.017185, y_c + -0.004661, z_c, rx, ry, rz], a, v)
    movel(p[x_c + 0.017192, y_c + -0.004515, z_c, rx, ry, rz], a, v)
    movel(p[x_c + 0.017199, y_c + -0.004370, z_c, rx, ry, rz], a, v)
    movel(p[x_c + 0.017206, y_c + -0.004225, z_c, rx, ry, rz], a, v)
    movel(p[x_c + 0.017213, y_c + -0.004081, z_c, rx, ry, rz], a, v)
    movel(p[x_c + 0.017219, y_c + -0.003938, z_c, rx, ry, rz], a, v)
    movel(p[x_c + 0.017225, y_c + -0.003796, z_c, rx, ry, rz], a, v)
    movel(p[x_c + 0.017231, y_c + -0.003655, z_c, rx, ry, rz], a, v)
    movel(p[x_c + 0.017236, y_c + -0.003515, z_c, rx, ry, rz], a, v)
    movel(p[x_c + 0.017242, y_c + -0.003376, z_c, rx, ry, rz], a, v)
    movel(p[x_c + 0.017247, y_c + -0.003239, z_c, rx, ry, rz], a, v)
    movel(p[x_c + 0.017251, y_c + -0.003104, z_c, rx, ry, rz], a, v)
    movel(p[x_c + 0.017255, y_c + -0.002970, z_c, rx, ry, rz], a, v)
    movel(p[x_c + 0.017259, y_c + -0.002838, z_c, rx, ry, rz], a, v)
    movel(p[x_c + 0.017263, y_c + -0.002708, z_c, rx, ry, rz], a, v)
    movel(p[x_c + 0.017266, y_c + -0.002579, z_c, rx, ry, rz], a, v)
    movel(p[x_c + 0.017270, y_c + -0.002453, z_c, rx, ry, rz], a, v)
    movel(p[x_c + 0.017272, y_c + -0.002329, z_c, rx, ry, rz], a, v)
    movel(p[x_c + 0.017275, y_c + -0.002207, z_c, rx, ry, rz], a, v)
    movel(p[x_c + 0.017277, y_c + -0.002087, z_c, rx, ry, rz], a, v)
    movel(p[x_c + 0.017279, y_c + -0.001970, z_c, rx, ry, rz], a, v)
    movel(p[x_c + 0.017280, y_c + -0.001855, z_c, rx, ry, rz], a, v)
    movel(p[x_c + 0.017281, y_c + -0.001743, z_c, rx, ry, rz], a, v)
    movel(p[x_c + 0.017282, y_c + -0.001634, z_c, rx, ry, rz], a, v)
    movel(p[x_c + 0.017283, y_c + -0.001527, z_c, rx, ry, rz], a, v)
    movel(p[x_c + 0.017283, y_c + -0.001424, z_c, rx, ry, rz], a, v)
    movel(p[x_c + 0.017283, y_c + -0.001323, z_c, rx, ry, rz], a, v)
    movel(p[x_c + 0.017282, y_c + -0.001226, z_c, rx, ry, rz], a, v)
    movel(p[x_c + 0.017282, y_c + -0.001131, z_c, rx, ry, rz], a, v)
    movel(p[x_c + 0.017280, y_c + -0.001040, z_c, rx, ry, rz], a, v)
    movel(p[x_c + 0.017279, y_c + -0.000953, z_c, rx, ry, rz], a, v)
    movel(p[x_c + 0.017277, y_c + -0.000869, z_c, rx, ry, rz], a, v)
    movel(p[x_c + 0.017275, y_c + -0.000788, z_c, rx, ry, rz], a, v)
    movel(p[x_c + 0.017272, y_c + -0.000712, z_c, rx, ry, rz], a, v)
    movel(p[x_c + 0.017270, y_c + -0.000639, z_c, rx, ry, rz], a, v)
    movel(p[x_c + 0.017266, y_c + -0.000570, z_c, rx, ry, rz], a, v)
    movel(p[x_c + 0.017263, y_c + -0.000505, z_c, rx, ry, rz], a, v)
    movel(p[x_c + 0.017259, y_c + -0.000444, z_c, rx, ry, rz], a, v)
    movel(p[x_c + 0.017255, y_c + -0.000388, z_c, rx, ry, rz], a, v)
    movel(p[x_c + 0.017250, y_c + -0.000336, z_c, rx, ry, rz], a, v)
    movel(p[x_c + 0.017245, y_c + -0.000288, z_c, rx, ry, rz], a, v)
    movel(p[x_c + 0.017240, y_c + -0.000245, z_c, rx, ry, rz], a, v)
    movel(p[x_c + 0.017240, y_c + -0.000245, z_c, rx, ry, rz], a, v)
    movel(p[x_c + 0.017227, y_c + -0.000153, z_c, rx, ry, rz], a, v)
    movel(p[x_c + 0.017213, y_c + -0.000063, z_c, rx, ry, rz], a, v)
    movel(p[x_c + 0.017200, y_c + 0.000025, z_c, rx, ry, rz], a, v)
    movel(p[x_c + 0.017185, y_c + 0.000112, z_c, rx, ry, rz], a, v)
    movel(p[x_c + 0.017169, y_c + 0.000198, z_c, rx, ry, rz], a, v)
    movel(p[x_c + 0.017153, y_c + 0.000283, z_c, rx, ry, rz], a, v)
    movel(p[x_c + 0.017136, y_c + 0.000367, z_c, rx, ry, rz], a, v)
    movel(p[x_c + 0.017117, y_c + 0.000450, z_c, rx, ry, rz], a, v)
    movel(p[x_c + 0.017098, y_c + 0.000534, z_c, rx, ry, rz], a, v)
    movel(p[x_c + 0.017077, y_c + 0.000617, z_c, rx, ry, rz], a, v)
    movel(p[x_c + 0.017054, y_c + 0.000699, z_c, rx, ry, rz], a, v)
    movel(p[x_c + 0.017030, y_c + 0.000783, z_c, rx, ry, rz], a, v)
    movel(p[x_c + 0.017004, y_c + 0.000866, z_c, rx, ry, rz], a, v)
    movel(p[x_c + 0.016977, y_c + 0.000951, z_c, rx, ry, rz], a, v)
    movel(p[x_c + 0.016948, y_c + 0.001036, z_c, rx, ry, rz], a, v)
    movel(p[x_c + 0.016917, y_c + 0.001122, z_c, rx, ry, rz], a, v)
    movel(p[x_c + 0.016884, y_c + 0.001209, z_c, rx, ry, rz], a, v)
    movel(p[x_c + 0.016848, y_c + 0.001298, z_c, rx, ry, rz], a, v)
    movel(p[x_c + 0.016811, y_c + 0.001389, z_c, rx, ry, rz], a, v)
    movel(p[x_c + 0.016771, y_c + 0.001481, z_c, rx, ry, rz], a, v)
    movel(p[x_c + 0.016728, y_c + 0.001575, z_c, rx, ry, rz], a, v)
    movel(p[x_c + 0.016684, y_c + 0.001672, z_c, rx, ry, rz], a, v)
    movel(p[x_c + 0.016636, y_c + 0.001771, z_c, rx, ry, rz], a, v)
    movel(p[x_c + 0.016586, y_c + 0.001873, z_c, rx, ry, rz], a, v)
    movel(p[x_c + 0.016532, y_c + 0.001977, z_c, rx, ry, rz], a, v)
    movel(p[x_c + 0.016476, y_c + 0.002085, z_c, rx, ry, rz], a, v)
    movel(p[x_c + 0.016417, y_c + 0.002196, z_c, rx, ry, rz], a, v)
    movel(p[x_c + 0.016354, y_c + 0.002311, z_c, rx, ry, rz], a, v)
    movel(p[x_c + 0.016289, y_c + 0.002429, z_c, rx, ry, rz], a, v)
    movel(p[x_c + 0.016220, y_c + 0.002551, z_c, rx, ry, rz], a, v)
    movel(p[x_c + 0.016147, y_c + 0.002677, z_c, rx, ry, rz], a, v)
    movel(p[x_c + 0.016071, y_c + 0.002807, z_c, rx, ry, rz], a, v)
    movel(p[x_c + 0.015991, y_c + 0.002942, z_c, rx, ry, rz], a, v)
    movel(p[x_c + 0.015908, y_c + 0.003081, z_c, rx, ry, rz], a, v)
    movel(p[x_c + 0.015820, y_c + 0.003226, z_c, rx, ry, rz], a, v)
    movel(p[x_c + 0.015729, y_c + 0.003375, z_c, rx, ry, rz], a, v)
    movel(p[x_c + 0.015633, y_c + 0.003530, z_c, rx, ry, rz], a, v)
    movel(p[x_c + 0.015533, y_c + 0.003690, z_c, rx, ry, rz], a, v)
    movel(p[x_c + 0.015429, y_c + 0.003856, z_c, rx, ry, rz], a, v)
    movel(p[x_c + 0.015321, y_c + 0.004028, z_c, rx, ry, rz], a, v)
    movel(p[x_c + 0.015208, y_c + 0.004205, z_c, rx, ry, rz], a, v)
    movel(p[x_c + 0.015090, y_c + 0.004390, z_c, rx, ry, rz], a, v)
    movel(p[x_c + 0.014968, y_c + 0.004580, z_c, rx, ry, rz], a, v)
    movel(p[x_c + 0.014840, y_c + 0.004778, z_c, rx, ry, rz], a, v)
    movel(p[x_c + 0.014708, y_c + 0.004982, z_c, rx, ry, rz], a, v)
    movel(p[x_c + 0.014571, y_c + 0.005193, z_c, rx, ry, rz], a, v)
    movel(p[x_c + 0.014429, y_c + 0.005412, z_c, rx, ry, rz], a, v)
    movel(p[x_c + 0.014282, y_c + 0.005638, z_c, rx, ry, rz], a, v)
    movel(p[x_c + 0.014129, y_c + 0.005872, z_c, rx, ry, rz], a, v)
    movel(p[x_c + 0.014129, y_c + 0.005872, z_c, rx, ry, rz], a, v)
    movel(p[x_c + 0.013909, y_c + 0.006211, z_c, rx, ry, rz], a, v)
    movel(p[x_c + 0.013691, y_c + 0.006549, z_c, rx, ry, rz], a, v)
    movel(p[x_c + 0.013477, y_c + 0.006888, z_c, rx, ry, rz], a, v)
    movel(p[x_c + 0.013264, y_c + 0.007228, z_c, rx, ry, rz], a, v)
    movel(p[x_c + 0.013055, y_c + 0.007568, z_c, rx, ry, rz], a, v)
    movel(p[x_c + 0.012847, y_c + 0.007908, z_c, rx, ry, rz], a, v)
    movel(p[x_c + 0.012643, y_c + 0.008249, z_c, rx, ry, rz], a, v)
    movel(p[x_c + 0.012440, y_c + 0.008590, z_c, rx, ry, rz], a, v)
    movel(p[x_c + 0.012240, y_c + 0.008932, z_c, rx, ry, rz], a, v)
    movel(p[x_c + 0.012043, y_c + 0.009275, z_c, rx, ry, rz], a, v)
    movel(p[x_c + 0.011847, y_c + 0.009619, z_c, rx, ry, rz], a, v)
    movel(p[x_c + 0.011654, y_c + 0.009964, z_c, rx, ry, rz], a, v)
    movel(p[x_c + 0.011464, y_c + 0.010309, z_c, rx, ry, rz], a, v)
    movel(p[x_c + 0.011275, y_c + 0.010656, z_c, rx, ry, rz], a, v)
    movel(p[x_c + 0.011089, y_c + 0.011004, z_c, rx, ry, rz], a, v)
    movel(p[x_c + 0.010905, y_c + 0.011352, z_c, rx, ry, rz], a, v)
    movel(p[x_c + 0.010723, y_c + 0.011703, z_c, rx, ry, rz], a, v)
    movel(p[x_c + 0.010544, y_c + 0.012054, z_c, rx, ry, rz], a, v)
    movel(p[x_c + 0.010366, y_c + 0.012407, z_c, rx, ry, rz], a, v)
    movel(p[x_c + 0.010190, y_c + 0.012761, z_c, rx, ry, rz], a, v)
    movel(p[x_c + 0.010017, y_c + 0.013117, z_c, rx, ry, rz], a, v)
    movel(p[x_c + 0.009845, y_c + 0.013474, z_c, rx, ry, rz], a, v)
    movel(p[x_c + 0.009676, y_c + 0.013833, z_c, rx, ry, rz], a, v)
    movel(p[x_c + 0.009508, y_c + 0.014194, z_c, rx, ry, rz], a, v)
    movel(p[x_c + 0.009342, y_c + 0.014556, z_c, rx, ry, rz], a, v)
    movel(p[x_c + 0.009178, y_c + 0.014920, z_c, rx, ry, rz], a, v)
    movel(p[x_c + 0.009016, y_c + 0.015286, z_c, rx, ry, rz], a, v)
    movel(p[x_c + 0.008856, y_c + 0.015655, z_c, rx, ry, rz], a, v)
    movel(p[x_c + 0.008697, y_c + 0.016025, z_c, rx, ry, rz], a, v)
    movel(p[x_c + 0.008541, y_c + 0.016397, z_c, rx, ry, rz], a, v)
    movel(p[x_c + 0.008386, y_c + 0.016772, z_c, rx, ry, rz], a, v)
    movel(p[x_c + 0.008232, y_c + 0.017148, z_c, rx, ry, rz], a, v)
    movel(p[x_c + 0.008081, y_c + 0.017527, z_c, rx, ry, rz], a, v)
    movel(p[x_c + 0.007931, y_c + 0.017909, z_c, rx, ry, rz], a, v)
    movel(p[x_c + 0.007782, y_c + 0.018293, z_c, rx, ry, rz], a, v)
    movel(p[x_c + 0.007635, y_c + 0.018679, z_c, rx, ry, rz], a, v)
    movel(p[x_c + 0.007490, y_c + 0.019068, z_c, rx, ry, rz], a, v)
    movel(p[x_c + 0.007346, y_c + 0.019460, z_c, rx, ry, rz], a, v)
    movel(p[x_c + 0.007204, y_c + 0.019854, z_c, rx, ry, rz], a, v)
    movel(p[x_c + 0.007063, y_c + 0.020251, z_c, rx, ry, rz], a, v)
    movel(p[x_c + 0.006924, y_c + 0.020651, z_c, rx, ry, rz], a, v)
    movel(p[x_c + 0.006785, y_c + 0.021054, z_c, rx, ry, rz], a, v)
    movel(p[x_c + 0.006649, y_c + 0.021460, z_c, rx, ry, rz], a, v)
    movel(p[x_c + 0.006513, y_c + 0.021869, z_c, rx, ry, rz], a, v)
    movel(p[x_c + 0.006379, y_c + 0.022281, z_c, rx, ry, rz], a, v)
    movel(p[x_c + 0.006246, y_c + 0.022696, z_c, rx, ry, rz], a, v)
    movel(p[x_c + 0.006114, y_c + 0.023115, z_c, rx, ry, rz], a, v)
    movel(p[x_c + 0.005984, y_c + 0.023537, z_c, rx, ry, rz], a, v)
    movel(p[x_c + 0.005854, y_c + 0.023962, z_c, rx, ry, rz], a, v)
    movel(p[x_c + 0.005854, y_c + 0.023962, z_c, rx, ry, rz], a, v)
    movel(p[x_c + 0.005769, y_c + 0.024247, z_c, rx, ry, rz], a, v)
    movel(p[x_c + 0.005685, y_c + 0.024526, z_c, rx, ry, rz], a, v)
    movel(p[x_c + 0.005603, y_c + 0.024801, z_c, rx, ry, rz], a, v)
    movel(p[x_c + 0.005522, y_c + 0.025073, z_c, rx, ry, rz], a, v)
    movel(p[x_c + 0.005443, y_c + 0.025341, z_c, rx, ry, rz], a, v)
    movel(p[x_c + 0.005366, y_c + 0.025605, z_c, rx, ry, rz], a, v)
    movel(p[x_c + 0.005289, y_c + 0.025868, z_c, rx, ry, rz], a, v)
    movel(p[x_c + 0.005214, y_c + 0.026128, z_c, rx, ry, rz], a, v)
    movel(p[x_c + 0.005140, y_c + 0.026386, z_c, rx, ry, rz], a, v)
    movel(p[x_c + 0.005067, y_c + 0.026643, z_c, rx, ry, rz], a, v)
    movel(p[x_c + 0.004994, y_c + 0.026899, z_c, rx, ry, rz], a, v)
    movel(p[x_c + 0.004922, y_c + 0.027155, z_c, rx, ry, rz], a, v)
    movel(p[x_c + 0.004851, y_c + 0.027411, z_c, rx, ry, rz], a, v)
    movel(p[x_c + 0.004781, y_c + 0.027667, z_c, rx, ry, rz], a, v)
    movel(p[x_c + 0.004710, y_c + 0.027925, z_c, rx, ry, rz], a, v)
    movel(p[x_c + 0.004640, y_c + 0.028184, z_c, rx, ry, rz], a, v)
    movel(p[x_c + 0.004570, y_c + 0.028445, z_c, rx, ry, rz], a, v)
    movel(p[x_c + 0.004500, y_c + 0.028708, z_c, rx, ry, rz], a, v)
    movel(p[x_c + 0.004430, y_c + 0.028973, z_c, rx, ry, rz], a, v)
    movel(p[x_c + 0.004360, y_c + 0.029242, z_c, rx, ry, rz], a, v)
    movel(p[x_c + 0.004290, y_c + 0.029515, z_c, rx, ry, rz], a, v)
    movel(p[x_c + 0.004219, y_c + 0.029792, z_c, rx, ry, rz], a, v)
    movel(p[x_c + 0.004147, y_c + 0.030073, z_c, rx, ry, rz], a, v)
    movel(p[x_c + 0.004075, y_c + 0.030360, z_c, rx, ry, rz], a, v)
    movel(p[x_c + 0.004002, y_c + 0.030652, z_c, rx, ry, rz], a, v)
    movel(p[x_c + 0.003929, y_c + 0.030949, z_c, rx, ry, rz], a, v)
    movel(p[x_c + 0.003854, y_c + 0.031253, z_c, rx, ry, rz], a, v)
    movel(p[x_c + 0.003778, y_c + 0.031564, z_c, rx, ry, rz], a, v)
    movel(p[x_c + 0.003701, y_c + 0.031882, z_c, rx, ry, rz], a, v)
    movel(p[x_c + 0.003623, y_c + 0.032208, z_c, rx, ry, rz], a, v)
    movel(p[x_c + 0.003543, y_c + 0.032542, z_c, rx, ry, rz], a, v)
    movel(p[x_c + 0.003462, y_c + 0.032884, z_c, rx, ry, rz], a, v)
    movel(p[x_c + 0.003379, y_c + 0.033236, z_c, rx, ry, rz], a, v)
    movel(p[x_c + 0.003295, y_c + 0.033597, z_c, rx, ry, rz], a, v)
    movel(p[x_c + 0.003208, y_c + 0.033968, z_c, rx, ry, rz], a, v)
    movel(p[x_c + 0.003120, y_c + 0.034349, z_c, rx, ry, rz], a, v)
    movel(p[x_c + 0.003029, y_c + 0.034741, z_c, rx, ry, rz], a, v)
    movel(p[x_c + 0.002936, y_c + 0.035144, z_c, rx, ry, rz], a, v)
    movel(p[x_c + 0.002841, y_c + 0.035559, z_c, rx, ry, rz], a, v)
    movel(p[x_c + 0.002744, y_c + 0.035987, z_c, rx, ry, rz], a, v)
    movel(p[x_c + 0.002644, y_c + 0.036426, z_c, rx, ry, rz], a, v)
    movel(p[x_c + 0.002541, y_c + 0.036879, z_c, rx, ry, rz], a, v)
    movel(p[x_c + 0.002436, y_c + 0.037346, z_c, rx, ry, rz], a, v)
    movel(p[x_c + 0.002327, y_c + 0.037826, z_c, rx, ry, rz], a, v)
    movel(p[x_c + 0.002216, y_c + 0.038320, z_c, rx, ry, rz], a, v)
    movel(p[x_c + 0.002102, y_c + 0.038830, z_c, rx, ry, rz], a, v)
    movel(p[x_c + 0.001984, y_c + 0.039355, z_c, rx, ry, rz], a, v)
    movel(p[x_c + 0.001863, y_c + 0.039895, z_c, rx, ry, rz], a, v)
    movel(p[x_c + 0.001739, y_c + 0.040452, z_c, rx, ry, rz], a, v)
    movel(p[x_c + 0.001739, y_c + 0.040452, z_c, rx, ry, rz], a, v)
    movel(p[x_c + 0.001577, y_c + 0.041177, z_c, rx, ry, rz], a, v)
    movel(p[x_c + 0.001419, y_c + 0.041879, z_c, rx, ry, rz], a, v)
    movel(p[x_c + 0.001266, y_c + 0.042558, z_c, rx, ry, rz], a, v)
    movel(p[x_c + 0.001118, y_c + 0.043216, z_c, rx, ry, rz], a, v)
    movel(p[x_c + 0.000973, y_c + 0.043853, z_c, rx, ry, rz], a, v)
    movel(p[x_c + 0.000832, y_c + 0.044469, z_c, rx, ry, rz], a, v)
    movel(p[x_c + 0.000695, y_c + 0.045064, z_c, rx, ry, rz], a, v)
    movel(p[x_c + 0.000561, y_c + 0.045641, z_c, rx, ry, rz], a, v)
    movel(p[x_c + 0.000431, y_c + 0.046198, z_c, rx, ry, rz], a, v)
    movel(p[x_c + 0.000304, y_c + 0.046737, z_c, rx, ry, rz], a, v)
    movel(p[x_c + 0.000180, y_c + 0.047258, z_c, rx, ry, rz], a, v)
    movel(p[x_c + 0.000059, y_c + 0.047763, z_c, rx, ry, rz], a, v)
    movel(p[x_c + -0.000059, y_c + 0.048250, z_c, rx, ry, rz], a, v)
    movel(p[x_c + -0.000175, y_c + 0.048722, z_c, rx, ry, rz], a, v)
    movel(p[x_c + -0.000289, y_c + 0.049178, z_c, rx, ry, rz], a, v)
    movel(p[x_c + -0.000400, y_c + 0.049619, z_c, rx, ry, rz], a, v)
    movel(p[x_c + -0.000509, y_c + 0.050046, z_c, rx, ry, rz], a, v)
    movel(p[x_c + -0.000617, y_c + 0.050459, z_c, rx, ry, rz], a, v)
    movel(p[x_c + -0.000723, y_c + 0.050860, z_c, rx, ry, rz], a, v)
    movel(p[x_c + -0.000828, y_c + 0.051247, z_c, rx, ry, rz], a, v)
    movel(p[x_c + -0.000931, y_c + 0.051623, z_c, rx, ry, rz], a, v)
    movel(p[x_c + -0.001033, y_c + 0.051987, z_c, rx, ry, rz], a, v)
    movel(p[x_c + -0.001134, y_c + 0.052341, z_c, rx, ry, rz], a, v)
    movel(p[x_c + -0.001234, y_c + 0.052684, z_c, rx, ry, rz], a, v)
    movel(p[x_c + -0.001334, y_c + 0.053018, z_c, rx, ry, rz], a, v)
    movel(p[x_c + -0.001433, y_c + 0.053343, z_c, rx, ry, rz], a, v)
    movel(p[x_c + -0.001532, y_c + 0.053659, z_c, rx, ry, rz], a, v)
    movel(p[x_c + -0.001631, y_c + 0.053967, z_c, rx, ry, rz], a, v)
    movel(p[x_c + -0.001731, y_c + 0.054268, z_c, rx, ry, rz], a, v)
    movel(p[x_c + -0.001830, y_c + 0.054563, z_c, rx, ry, rz], a, v)
    movel(p[x_c + -0.001930, y_c + 0.054851, z_c, rx, ry, rz], a, v)
    movel(p[x_c + -0.002030, y_c + 0.055133, z_c, rx, ry, rz], a, v)
    movel(p[x_c + -0.002131, y_c + 0.055411, z_c, rx, ry, rz], a, v)
    movel(p[x_c + -0.002234, y_c + 0.055684, z_c, rx, ry, rz], a, v)
    movel(p[x_c + -0.002337, y_c + 0.055954, z_c, rx, ry, rz], a, v)
    movel(p[x_c + -0.002441, y_c + 0.056220, z_c, rx, ry, rz], a, v)
    movel(p[x_c + -0.002548, y_c + 0.056483, z_c, rx, ry, rz], a, v)
    movel(p[x_c + -0.002655, y_c + 0.056745, z_c, rx, ry, rz], a, v)
    movel(p[x_c + -0.002765, y_c + 0.057004, z_c, rx, ry, rz], a, v)
    movel(p[x_c + -0.002876, y_c + 0.057263, z_c, rx, ry, rz], a, v)
    movel(p[x_c + -0.002990, y_c + 0.057522, z_c, rx, ry, rz], a, v)
    movel(p[x_c + -0.003106, y_c + 0.057781, z_c, rx, ry, rz], a, v)
    movel(p[x_c + -0.003225, y_c + 0.058040, z_c, rx, ry, rz], a, v)
    movel(p[x_c + -0.003346, y_c + 0.058301, z_c, rx, ry, rz], a, v)
    movel(p[x_c + -0.003470, y_c + 0.058564, z_c, rx, ry, rz], a, v)
    movel(p[x_c + -0.003598, y_c + 0.058830, z_c, rx, ry, rz], a, v)
    movel(p[x_c + -0.003728, y_c + 0.059099, z_c, rx, ry, rz], a, v)
    movel(p[x_c + -0.003862, y_c + 0.059371, z_c, rx, ry, rz], a, v)
    movel(p[x_c + -0.003999, y_c + 0.059648, z_c, rx, ry, rz], a, v)
    movel(p[x_c + -0.003999, y_c + 0.059648, z_c, rx, ry, rz], a, v)
    movel(p[x_c + -0.004178, y_c + 0.060001, z_c, rx, ry, rz], a, v)
    movel(p[x_c + -0.004359, y_c + 0.060350, z_c, rx, ry, rz], a, v)
    movel(p[x_c + -0.004542, y_c + 0.060695, z_c, rx, ry, rz], a, v)
    movel(p[x_c + -0.004729, y_c + 0.061036, z_c, rx, ry, rz], a, v)
    movel(p[x_c + -0.004917, y_c + 0.061373, z_c, rx, ry, rz], a, v)
    movel(p[x_c + -0.005109, y_c + 0.061707, z_c, rx, ry, rz], a, v)
    movel(p[x_c + -0.005303, y_c + 0.062037, z_c, rx, ry, rz], a, v)
    movel(p[x_c + -0.005499, y_c + 0.062362, z_c, rx, ry, rz], a, v)
    movel(p[x_c + -0.005698, y_c + 0.062684, z_c, rx, ry, rz], a, v)
    movel(p[x_c + -0.005899, y_c + 0.063001, z_c, rx, ry, rz], a, v)
    movel(p[x_c + -0.006103, y_c + 0.063315, z_c, rx, ry, rz], a, v)
    movel(p[x_c + -0.006310, y_c + 0.063625, z_c, rx, ry, rz], a, v)
    movel(p[x_c + -0.006519, y_c + 0.063931, z_c, rx, ry, rz], a, v)
    movel(p[x_c + -0.006730, y_c + 0.064232, z_c, rx, ry, rz], a, v)
    movel(p[x_c + -0.006944, y_c + 0.064530, z_c, rx, ry, rz], a, v)
    movel(p[x_c + -0.007160, y_c + 0.064823, z_c, rx, ry, rz], a, v)
    movel(p[x_c + -0.007379, y_c + 0.065113, z_c, rx, ry, rz], a, v)
    movel(p[x_c + -0.007600, y_c + 0.065398, z_c, rx, ry, rz], a, v)
    movel(p[x_c + -0.007823, y_c + 0.065679, z_c, rx, ry, rz], a, v)
    movel(p[x_c + -0.008049, y_c + 0.065956, z_c, rx, ry, rz], a, v)
    movel(p[x_c + -0.008277, y_c + 0.066229, z_c, rx, ry, rz], a, v)
    movel(p[x_c + -0.008507, y_c + 0.066498, z_c, rx, ry, rz], a, v)
    movel(p[x_c + -0.008740, y_c + 0.066763, z_c, rx, ry, rz], a, v)
    movel(p[x_c + -0.008975, y_c + 0.067023, z_c, rx, ry, rz], a, v)
    movel(p[x_c + -0.009213, y_c + 0.067280, z_c, rx, ry, rz], a, v)
    movel(p[x_c + -0.009452, y_c + 0.067532, z_c, rx, ry, rz], a, v)
    movel(p[x_c + -0.009694, y_c + 0.067780, z_c, rx, ry, rz], a, v)
    movel(p[x_c + -0.009939, y_c + 0.068023, z_c, rx, ry, rz], a, v)
    movel(p[x_c + -0.010185, y_c + 0.068263, z_c, rx, ry, rz], a, v)
    movel(p[x_c + -0.010434, y_c + 0.068498, z_c, rx, ry, rz], a, v)
    movel(p[x_c + -0.010685, y_c + 0.068729, z_c, rx, ry, rz], a, v)
    movel(p[x_c + -0.010938, y_c + 0.068955, z_c, rx, ry, rz], a, v)
    movel(p[x_c + -0.011193, y_c + 0.069177, z_c, rx, ry, rz], a, v)
    movel(p[x_c + -0.011451, y_c + 0.069395, z_c, rx, ry, rz], a, v)
    movel(p[x_c + -0.011710, y_c + 0.069609, z_c, rx, ry, rz], a, v)
    movel(p[x_c + -0.011972, y_c + 0.069818, z_c, rx, ry, rz], a, v)
    movel(p[x_c + -0.012236, y_c + 0.070023, z_c, rx, ry, rz], a, v)
    movel(p[x_c + -0.012502, y_c + 0.070223, z_c, rx, ry, rz], a, v)
    movel(p[x_c + -0.012770, y_c + 0.070419, z_c, rx, ry, rz], a, v)
    movel(p[x_c + -0.013040, y_c + 0.070611, z_c, rx, ry, rz], a, v)
    movel(p[x_c + -0.013313, y_c + 0.070798, z_c, rx, ry, rz], a, v)
    movel(p[x_c + -0.013587, y_c + 0.070981, z_c, rx, ry, rz], a, v)
    movel(p[x_c + -0.013864, y_c + 0.071159, z_c, rx, ry, rz], a, v)
    movel(p[x_c + -0.014142, y_c + 0.071333, z_c, rx, ry, rz], a, v)
    movel(p[x_c + -0.014423, y_c + 0.071502, z_c, rx, ry, rz], a, v)
    movel(p[x_c + -0.014705, y_c + 0.071667, z_c, rx, ry, rz], a, v)
    movel(p[x_c + -0.014990, y_c + 0.071827, z_c, rx, ry, rz], a, v)
    movel(p[x_c + -0.015276, y_c + 0.071983, z_c, rx, ry, rz], a, v)
    movel(p[x_c + -0.015565, y_c + 0.072134, z_c, rx, ry, rz], a, v)
    movel(p[x_c + -0.015565, y_c + 0.072134, z_c, rx, ry, rz], a, v)
    movel(p[x_c + -0.015717, y_c + 0.072212, z_c, rx, ry, rz], a, v)
    movel(p[x_c + -0.015869, y_c + 0.072288, z_c, rx, ry, rz], a, v)
    movel(p[x_c + -0.016018, y_c + 0.072362, z_c, rx, ry, rz], a, v)
    movel(p[x_c + -0.016167, y_c + 0.072435, z_c, rx, ry, rz], a, v)
    movel(p[x_c + -0.016314, y_c + 0.072506, z_c, rx, ry, rz], a, v)
    movel(p[x_c + -0.016461, y_c + 0.072575, z_c, rx, ry, rz], a, v)
    movel(p[x_c + -0.016606, y_c + 0.072643, z_c, rx, ry, rz], a, v)
    movel(p[x_c + -0.016750, y_c + 0.072709, z_c, rx, ry, rz], a, v)
    movel(p[x_c + -0.016894, y_c + 0.072773, z_c, rx, ry, rz], a, v)
    movel(p[x_c + -0.017036, y_c + 0.072835, z_c, rx, ry, rz], a, v)
    movel(p[x_c + -0.017178, y_c + 0.072896, z_c, rx, ry, rz], a, v)
    movel(p[x_c + -0.017319, y_c + 0.072956, z_c, rx, ry, rz], a, v)
    movel(p[x_c + -0.017460, y_c + 0.073014, z_c, rx, ry, rz], a, v)
    movel(p[x_c + -0.017600, y_c + 0.073070, z_c, rx, ry, rz], a, v)
    movel(p[x_c + -0.017740, y_c + 0.073125, z_c, rx, ry, rz], a, v)
    movel(p[x_c + -0.017880, y_c + 0.073179, z_c, rx, ry, rz], a, v)
    movel(p[x_c + -0.018019, y_c + 0.073231, z_c, rx, ry, rz], a, v)
    movel(p[x_c + -0.018158, y_c + 0.073281, z_c, rx, ry, rz], a, v)
    movel(p[x_c + -0.018297, y_c + 0.073331, z_c, rx, ry, rz], a, v)
    movel(p[x_c + -0.018436, y_c + 0.073378, z_c, rx, ry, rz], a, v)
    movel(p[x_c + -0.018575, y_c + 0.073425, z_c, rx, ry, rz], a, v)
    movel(p[x_c + -0.018714, y_c + 0.073470, z_c, rx, ry, rz], a, v)
    movel(p[x_c + -0.018854, y_c + 0.073514, z_c, rx, ry, rz], a, v)
    movel(p[x_c + -0.018994, y_c + 0.073557, z_c, rx, ry, rz], a, v)
    movel(p[x_c + -0.019134, y_c + 0.073598, z_c, rx, ry, rz], a, v)
    movel(p[x_c + -0.019274, y_c + 0.073638, z_c, rx, ry, rz], a, v)
    movel(p[x_c + -0.019416, y_c + 0.073677, z_c, rx, ry, rz], a, v)
    movel(p[x_c + -0.019558, y_c + 0.073714, z_c, rx, ry, rz], a, v)
    movel(p[x_c + -0.019700, y_c + 0.073751, z_c, rx, ry, rz], a, v)
    movel(p[x_c + -0.019843, y_c + 0.073786, z_c, rx, ry, rz], a, v)
    movel(p[x_c + -0.019988, y_c + 0.073820, z_c, rx, ry, rz], a, v)
    movel(p[x_c + -0.020133, y_c + 0.073854, z_c, rx, ry, rz], a, v)
    movel(p[x_c + -0.020279, y_c + 0.073886, z_c, rx, ry, rz], a, v)
    movel(p[x_c + -0.020426, y_c + 0.073917, z_c, rx, ry, rz], a, v)
    movel(p[x_c + -0.020575, y_c + 0.073947, z_c, rx, ry, rz], a, v)
    movel(p[x_c + -0.020725, y_c + 0.073976, z_c, rx, ry, rz], a, v)
    movel(p[x_c + -0.020876, y_c + 0.074004, z_c, rx, ry, rz], a, v)
    movel(p[x_c + -0.021028, y_c + 0.074031, z_c, rx, ry, rz], a, v)
    movel(p[x_c + -0.021182, y_c + 0.074057, z_c, rx, ry, rz], a, v)
    movel(p[x_c + -0.021338, y_c + 0.074082, z_c, rx, ry, rz], a, v)
    movel(p[x_c + -0.021495, y_c + 0.074106, z_c, rx, ry, rz], a, v)
    movel(p[x_c + -0.021654, y_c + 0.074130, z_c, rx, ry, rz], a, v)
    movel(p[x_c + -0.021815, y_c + 0.074152, z_c, rx, ry, rz], a, v)
    movel(p[x_c + -0.021978, y_c + 0.074174, z_c, rx, ry, rz], a, v)
    movel(p[x_c + -0.022143, y_c + 0.074195, z_c, rx, ry, rz], a, v)
    movel(p[x_c + -0.022310, y_c + 0.074216, z_c, rx, ry, rz], a, v)
    movel(p[x_c + -0.022479, y_c + 0.074235, z_c, rx, ry, rz], a, v)
    movel(p[x_c + -0.022650, y_c + 0.074254, z_c, rx, ry, rz], a, v)
    movel(p[x_c + -0.022824, y_c + 0.074272, z_c, rx, ry, rz], a, v)
    movel(p[x_c + -0.022824, y_c + 0.074272, z_c, rx, ry, rz], a, v)
    movel(p[x_c + -0.023073, y_c + 0.074296, z_c, rx, ry, rz], a, v)
    movel(p[x_c + -0.023322, y_c + 0.074317, z_c, rx, ry, rz], a, v)
    movel(p[x_c + -0.023571, y_c + 0.074336, z_c, rx, ry, rz], a, v)
    movel(p[x_c + -0.023820, y_c + 0.074352, z_c, rx, ry, rz], a, v)
    movel(p[x_c + -0.024069, y_c + 0.074365, z_c, rx, ry, rz], a, v)
    movel(p[x_c + -0.024318, y_c + 0.074376, z_c, rx, ry, rz], a, v)
    movel(p[x_c + -0.024566, y_c + 0.074384, z_c, rx, ry, rz], a, v)
    movel(p[x_c + -0.024815, y_c + 0.074389, z_c, rx, ry, rz], a, v)
    movel(p[x_c + -0.025064, y_c + 0.074391, z_c, rx, ry, rz], a, v)
    movel(p[x_c + -0.025313, y_c + 0.074391, z_c, rx, ry, rz], a, v)
    movel(p[x_c + -0.025562, y_c + 0.074388, z_c, rx, ry, rz], a, v)
    movel(p[x_c + -0.025811, y_c + 0.074383, z_c, rx, ry, rz], a, v)
    movel(p[x_c + -0.026060, y_c + 0.074374, z_c, rx, ry, rz], a, v)
    movel(p[x_c + -0.026308, y_c + 0.074364, z_c, rx, ry, rz], a, v)
    movel(p[x_c + -0.026557, y_c + 0.074350, z_c, rx, ry, rz], a, v)
    movel(p[x_c + -0.026806, y_c + 0.074334, z_c, rx, ry, rz], a, v)
    movel(p[x_c + -0.027054, y_c + 0.074315, z_c, rx, ry, rz], a, v)
    movel(p[x_c + -0.027303, y_c + 0.074293, z_c, rx, ry, rz], a, v)
    movel(p[x_c + -0.027551, y_c + 0.074269, z_c, rx, ry, rz], a, v)
    movel(p[x_c + -0.027800, y_c + 0.074242, z_c, rx, ry, rz], a, v)
    movel(p[x_c + -0.028048, y_c + 0.074212, z_c, rx, ry, rz], a, v)
    movel(p[x_c + -0.028296, y_c + 0.074180, z_c, rx, ry, rz], a, v)
    movel(p[x_c + -0.028544, y_c + 0.074145, z_c, rx, ry, rz], a, v)
    movel(p[x_c + -0.028792, y_c + 0.074107, z_c, rx, ry, rz], a, v)
    movel(p[x_c + -0.029040, y_c + 0.074067, z_c, rx, ry, rz], a, v)
    movel(p[x_c + -0.029288, y_c + 0.074024, z_c, rx, ry, rz], a, v)
    movel(p[x_c + -0.029536, y_c + 0.073978, z_c, rx, ry, rz], a, v)
    movel(p[x_c + -0.029784, y_c + 0.073930, z_c, rx, ry, rz], a, v)
    movel(p[x_c + -0.030032, y_c + 0.073879, z_c, rx, ry, rz], a, v)
    movel(p[x_c + -0.030279, y_c + 0.073825, z_c, rx, ry, rz], a, v)
    movel(p[x_c + -0.030527, y_c + 0.073769, z_c, rx, ry, rz], a, v)
    movel(p[x_c + -0.030774, y_c + 0.073710, z_c, rx, ry, rz], a, v)
    movel(p[x_c + -0.031022, y_c + 0.073648, z_c, rx, ry, rz], a, v)
    movel(p[x_c + -0.031269, y_c + 0.073584, z_c, rx, ry, rz], a, v)
    movel(p[x_c + -0.031516, y_c + 0.073517, z_c, rx, ry, rz], a, v)
    movel(p[x_c + -0.031763, y_c + 0.073447, z_c, rx, ry, rz], a, v)
    movel(p[x_c + -0.032010, y_c + 0.073375, z_c, rx, ry, rz], a, v)
    movel(p[x_c + -0.032257, y_c + 0.073299, z_c, rx, ry, rz], a, v)
    movel(p[x_c + -0.032503, y_c + 0.073222, z_c, rx, ry, rz], a, v)
    movel(p[x_c + -0.032750, y_c + 0.073141, z_c, rx, ry, rz], a, v)
    movel(p[x_c + -0.032996, y_c + 0.073058, z_c, rx, ry, rz], a, v)
    movel(p[x_c + -0.033243, y_c + 0.072972, z_c, rx, ry, rz], a, v)
    movel(p[x_c + -0.033489, y_c + 0.072884, z_c, rx, ry, rz], a, v)
    movel(p[x_c + -0.033735, y_c + 0.072793, z_c, rx, ry, rz], a, v)
    movel(p[x_c + -0.033981, y_c + 0.072699, z_c, rx, ry, rz], a, v)
    movel(p[x_c + -0.034227, y_c + 0.072603, z_c, rx, ry, rz], a, v)
    movel(p[x_c + -0.034472, y_c + 0.072504, z_c, rx, ry, rz], a, v)
    movel(p[x_c + -0.034718, y_c + 0.072402, z_c, rx, ry, rz], a, v)
    movel(p[x_c + -0.034963, y_c + 0.072298, z_c, rx, ry, rz], a, v)
    movel(p[x_c + -0.034963, y_c + 0.072298, z_c, rx, ry, rz], a, v)
    movel(p[x_c + -0.035306, y_c + 0.072146, z_c, rx, ry, rz], a, v)
    movel(p[x_c + -0.035646, y_c + 0.071989, z_c, rx, ry, rz], a, v)
    movel(p[x_c + -0.035984, y_c + 0.071825, z_c, rx, ry, rz], a, v)
    movel(p[x_c + -0.036320, y_c + 0.071655, z_c, rx, ry, rz], a, v)
    movel(p[x_c + -0.036653, y_c + 0.071480, z_c, rx, ry, rz], a, v)
    movel(p[x_c + -0.036983, y_c + 0.071298, z_c, rx, ry, rz], a, v)
    movel(p[x_c + -0.037311, y_c + 0.071110, z_c, rx, ry, rz], a, v)
    movel(p[x_c + -0.037637, y_c + 0.070916, z_c, rx, ry, rz], a, v)
